RoboDK station: kr30 cnc 072119 yaaaasss.rdk

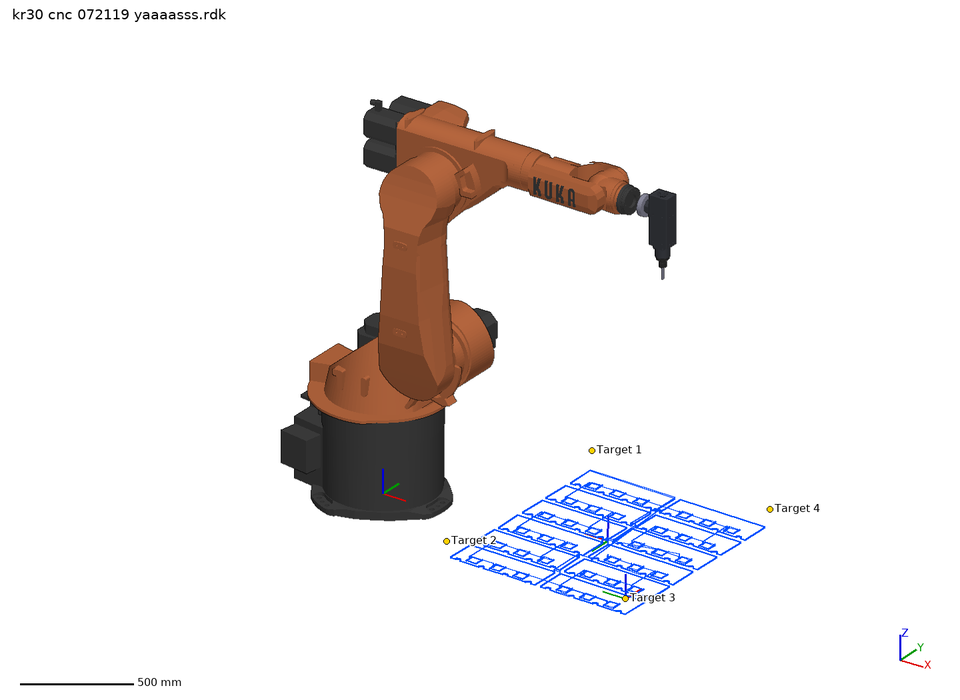
[picture v0: the station drawn from its stored meshes, robots at their saved joint values, targets as dots, program paths as lines]
Station kr30 cnc 072119 yaaaasss. Poses are relative to the parent item; angles as X-Y-Z fixed-axis rotations.
  - frame GIGASHEEN Base at (0, 0, 0) mm
    - robot GIGASHEEN (model KUKA KR 30 HA): 6 axes, payload 30 kg, reach 2033 mm, repeatability 0.05 mm, weight 665 kg
        modified DH rows (alpha deg, a mm, theta deg, d mm): 0, 0, 0, 815; -90, 350, 0, 0; 0, 850, -90, 0; -90, 145, 0, 820; 90, 0, 0, 0; -90, 0, 180, 170
        joint limits [-185, -135, -120, -350, -119, -350] to [185, 35, 158, 350, 119, 350]; home [0, -90, 90, 0, 0, 0]; saved at [0, -90, 90, 0, 0, 0]
      - tool 1/2" End Mill TCP, TCP at (337.71, -2.2, 160.57) mm, rotated rx 0 ry 90 rz 0 deg, size 415.8 x 102 x 153.6 mm
    - target Target 1 (joint target) at (982.46, 202.21, 406.25) mm, rotated rx -179.95 ry 0.15 rz -89.48 deg; joints [7.49, -59.642, 144.935, 97.969, -90.801, -4.608] of GIGASHEEN
    - target Target 2 (joint target) at (986.83, -921.64, 412.07) mm, rotated rx -179.94 ry 0.15 rz -89.48 deg; joints [51.766, -38.608, 94.384, 136.851, -116.554, -22.567] of GIGASHEEN
    - target Target 3 (joint target) at (1949.02, -919.97, 396.91) mm, rotated rx -179.94 ry 0.14 rz 179.61 deg; joints [29.5, -22.76, 62.288, 41.088, -47.759, -30.404] of GIGASHEEN
    - target Target 4 (joint target) at (1949.02, 190.94, 391.63) mm, rotated rx -179.94 ry 0.14 rz 179.61 deg; joints [-6.898, -35.989, 90.741, -8.88, -55.221, 5.167] of GIGASHEEN
  - machining project Machining Settings: C:/Users/liqui/OneDrive/Desktop/first half pipe jig.apt | rotZ(0) | rotX(0)*rotY(0) | rotZ(0)
  - program Prog2 (4 instructions, listed below)
  - frame Table at (1949.02, -919.97, 396.91) mm, rotated rx 0.87 ry 0.27 rz 90 deg
    - frame Frame 4 at (550, 480, -75) mm, rotated rx 0 ry 0 rz 90 deg
  - program Machining (1954 instructions, listed below)
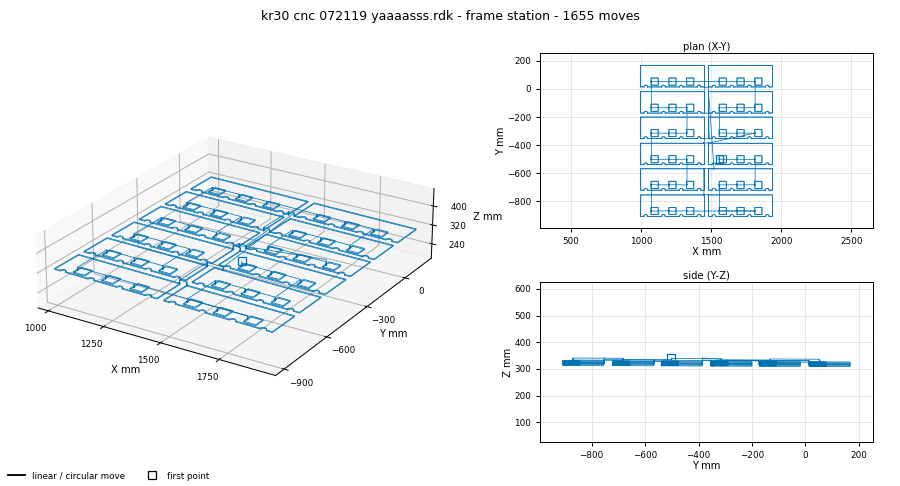
[picture p0: tool path of kr30 cnc 072119 yaaaasss.rdk in frame station, 1655 of 1659 moves have a stored position in this frame; points joined in program order, loops and branches not executed]

--- program Prog2 (robot GIGASHEEN) ---
  MoveJ (plywood back right safe) [its target is no longer in the station]
  MoveL (plywood back left safe) [its target is no longer in the station]
  MoveL (plywood front left safe) [its target is no longer in the station]
  MoveL (plywood front right safe) [its target is no longer in the station]

--- program Machining (robot GIGASHEEN) ---
  Smooth(1)
  Set Ref.: Frame 4
  Set Tool: 1/2" End Mill TCP
  Show 1/2" End Mill TCP
  Print: /'1001'
  Print: /''
  Print: /'2D Contour2'
  Set speed (1000.0 mm/s)
  MoveJ 1 to (-92.16, 131.48, 15) mm, rotated rx 180 ry 0 rz 0 deg; joints [21.959, -45.515, 117.936, 23.028, -72.87, -6.513]
  MoveL 2 to (-92.16, 131.48, 15) mm, rotated rx 180 ry 0 rz 0 deg; joints [21.959, -45.515, 117.936, 23.028, -72.87, -6.513]
  MoveL 3 to (-92.16, 131.48, 15) mm, rotated rx 180 ry 0 rz 0 deg; joints [21.959, -45.515, 117.936, 23.028, -72.87, -6.513]
  Set speed (1000.0 mm/s)
  MoveL 4 to (-92.16, 131.49, 6) mm, rotated rx -180 ry 0 rz 0 deg; joints [21.962, -44.952, 117.841, 22.976, -73.301, -6.323]
  Set speed (25.4 mm/s)
  MoveL 5 to (-92.16, 131.49, -3.54) mm, rotated rx -180 ry 0 rz 0 deg; joints [21.967, -44.354, 117.733, 22.924, -73.753, -6.125]
  MoveC 6 to (-91.98, 131.49, -3.99) mm, rotated rx -180 ry 0 rz 0 deg; joints [21.97, -44.331, 117.743, 22.924, -73.782, -6.113] to (-91.53, 131.48, -4.17) mm, rotated rx 180 ry 0 rz 0 deg; joints [21.977, -44.333, 117.775, 22.928, -73.811, -6.103]
  Set speed (50.8 mm/s)
  MoveL 7 to (-90.89, 131.48, -4.18) mm, rotated rx 180 ry 0 rz 0 deg; joints [21.987, -44.352, 117.824, 22.935, -73.84, -6.093]
  MoveC 8 to (-90.44, 131.3, -4.18) mm, rotated rx -180 ry 0 rz 0 deg; joints [21.987, -44.368, 117.865, 22.932, -73.863, -6.083] to (-90.26, 130.85, -4.18) mm, rotated rx -180 ry 0 rz 0 deg; joints [21.972, -44.379, 117.893, 22.915, -73.877, -6.072]
  MoveL 9 to (-90.26, 105.45, -4.17) mm, rotated rx -180 ry 0 rz 0 deg; joints [20.95, -44.663, 118.664, 21.805, -74.218, -5.605]
  MoveL 10 to (-141.06, 105.45, -4.17) mm, rotated rx -180 ry 0 rz 0 deg; joints [20.189, -43.084, 114.66, 21.285, -71.881, -6.316]
  MoveL 11 to (-141.06, 156.25, -4.17) mm, rotated rx -180 ry 0 rz 0 deg; joints [22.16, -42.482, 113.093, 23.47, -71.231, -7.326]
  MoveL 12 to (-90.26, 156.25, -4.17) mm, rotated rx 180 ry 0 rz 0 deg; joints [22.98, -44.078, 117.084, 24.017, -73.527, -6.56]
  MoveL 13 to (-90.26, 130.85, -4.18) mm, rotated rx -180 ry 0 rz 0 deg; joints [21.972, -44.379, 117.893, 22.915, -73.877, -6.072]
  MoveC 14 to (-90.44, 130.4, -4.17) mm, rotated rx -180 ry 0 rz 0 deg; joints [21.951, -44.379, 117.893, 22.893, -73.875, -6.066] to (-90.89, 130.21, -4.18) mm, rotated rx 180 ry 0 rz 0 deg; joints [21.937, -44.367, 117.864, 22.88, -73.857, -6.069]
  MoveL 15 to (-91.53, 130.21, -4.18) mm, rotated rx 180 ry 0 rz 0 deg; joints [21.926, -44.348, 117.815, 22.873, -73.829, -6.079]
  MoveC 16 to (-91.98, 130.21, -3.99) mm, rotated rx 180 ry 0 rz 0 deg; joints [21.919, -44.346, 117.782, 22.869, -73.8, -6.089] to (-92.16, 130.21, -3.54) mm, rotated rx -180 ry 0 rz 0 deg; joints [21.916, -44.368, 117.773, 22.869, -73.77, -6.101]
  Set speed (1000.0 mm/s)
  MoveL 17 to (-92.16, 130.21, 5) mm, rotated rx -180 ry 0 rz 0 deg; joints [21.912, -44.904, 117.87, 22.915, -73.365, -6.278]
  MoveL 18 to (-92.16, 131.48, 5) mm, rotated rx -180 ry 0 rz 0 deg; joints [21.963, -44.89, 117.83, 22.971, -73.348, -6.302]
  Set speed (25.4 mm/s)
  MoveL 19 to (-92.16, 131.49, 1.83) mm, rotated rx -180 ry 0 rz 0 deg; joints [21.964, -44.691, 117.795, 22.953, -73.499, -6.236]
  MoveL 20 to (-92.16, 131.49, -7.71) mm, rotated rx 180 ry 0 rz 0 deg; joints [21.968, -44.091, 117.684, 22.902, -73.949, -6.039]
  MoveC 21 to (-91.98, 131.48, -8.16) mm, rotated rx 180 ry 0 rz 0 deg; joints [21.972, -44.069, 117.693, 22.902, -73.979, -6.027] to (-91.53, 131.48, -8.35) mm, rotated rx 180 ry 0 rz 0 deg; joints [21.979, -44.07, 117.725, 22.906, -74.008, -6.017]
  Set speed (50.8 mm/s)
  MoveL 22 to (-90.89, 131.48, -8.35) mm, rotated rx 180 ry 0 rz 0 deg; joints [21.989, -44.089, 117.774, 22.913, -74.037, -6.007]
  MoveC 23 to (-90.44, 131.3, -8.35) mm, rotated rx 180 ry 0 rz 0 deg; joints [21.989, -44.105, 117.815, 22.91, -74.059, -5.997] to (-90.26, 130.85, -8.35) mm, rotated rx -180 ry 0 rz 0 deg; joints [21.974, -44.116, 117.843, 22.893, -74.074, -5.986]
  MoveL 24 to (-90.26, 105.45, -8.35) mm, rotated rx -180 ry 0 rz 0 deg; joints [20.951, -44.398, 118.614, 21.784, -74.418, -5.522]
  MoveL 25 to (-141.06, 105.45, -8.35) mm, rotated rx 180 ry 0 rz 0 deg; joints [20.191, -42.829, 114.611, 21.263, -72.072, -6.238]
  MoveL 26 to (-141.06, 156.25, -8.35) mm, rotated rx 180 ry 0 rz 0 deg; joints [22.162, -42.232, 113.044, 23.445, -71.416, -7.242]
  MoveL 27 to (-90.26, 156.25, -8.35) mm, rotated rx 180 ry 0 rz 0 deg; joints [22.982, -43.817, 117.034, 23.994, -73.72, -6.471]
  MoveL 28 to (-90.26, 130.85, -8.35) mm, rotated rx -180 ry 0 rz 0 deg; joints [21.974, -44.116, 117.843, 22.893, -74.074, -5.986]
  MoveC 29 to (-90.44, 130.4, -8.35) mm, rotated rx 180 ry 0 rz 0 deg; joints [21.953, -44.115, 117.843, 22.871, -74.072, -5.981] to (-90.89, 130.21, -8.35) mm, rotated rx 180 ry 0 rz 0 deg; joints [21.938, -44.104, 117.814, 22.858, -74.054, -5.984]
  MoveL 30 to (-91.53, 130.21, -8.35) mm, rotated rx 180 ry 0 rz 0 deg; joints [21.928, -44.085, 117.765, 22.851, -74.025, -5.993]
  MoveC 31 to (-91.98, 130.21, -8.16) mm, rotated rx -180 ry 0 rz 0 deg; joints [21.921, -44.083, 117.732, 22.847, -73.996, -6.004] to (-92.16, 130.22, -7.72) mm, rotated rx -180 ry 0 rz 0 deg; joints [21.918, -44.106, 117.723, 22.847, -73.966, -6.015]
  Set speed (1000.0 mm/s)
  MoveL 32 to (-92.16, 130.21, 6) mm, rotated rx -180 ry 0 rz 0 deg; joints [21.912, -44.967, 117.881, 22.921, -73.318, -6.299]
  MoveL 33 to (-219.16, 131.48, 6) mm, rotated rx 180 ry 0 rz 0 deg; joints [20.086, -40.721, 107.569, 21.82, -67.469, -8.132]
  Set speed (25.4 mm/s)
  MoveL 34 to (-219.16, 131.48, -3.54) mm, rotated rx -180 ry 0 rz 0 deg; joints [20.089, -40.181, 107.465, 21.757, -67.874, -7.958]
  MoveC 35 to (-218.98, 131.48, -3.99) mm, rotated rx 180 ry 0 rz 0 deg; joints [20.092, -40.162, 107.476, 21.756, -67.902, -7.948] to (-218.53, 131.49, -4.17) mm, rotated rx -180 ry 0 rz 0 deg; joints [20.098, -40.168, 107.512, 21.758, -67.931, -7.938]
  Set speed (50.8 mm/s)
  MoveL 36 to (-217.89, 131.48, -4.17) mm, rotated rx 180 ry 0 rz 0 deg; joints [20.107, -40.19, 107.565, 21.762, -67.962, -7.929]
  MoveC 37 to (-217.44, 131.3, -4.18) mm, rotated rx 180 ry 0 rz 0 deg; joints [20.106, -40.208, 107.609, 21.758, -67.985, -7.918] to (-217.26, 130.85, -4.18) mm, rotated rx -180 ry 0 rz 0 deg; joints [20.092, -40.22, 107.638, 21.74, -67.999, -7.906]
  MoveL 38 to (-217.26, 105.45, -4.18) mm, rotated rx 180 ry 0 rz 0 deg; joints [19.142, -40.524, 108.399, 20.66, -68.295, -7.365]
  MoveL 39 to (-268.06, 105.45, -4.18) mm, rotated rx 180 ry 0 rz 0 deg; joints [18.501, -38.685, 104.03, 20.345, -65.836, -8.068]
  MoveL 40 to (-268.06, 156.25, -4.18) mm, rotated rx -180 ry 0 rz 0 deg; joints [20.336, -38.042, 102.464, 22.49, -65.261, -9.235]
  MoveL 41 to (-217.26, 156.25, -4.17) mm, rotated rx -180 ry 0 rz 0 deg; joints [21.03, -39.899, 106.838, 22.816, -67.694, -8.465]
  MoveL 42 to (-217.26, 130.85, -4.18) mm, rotated rx -180 ry 0 rz 0 deg; joints [20.092, -40.22, 107.638, 21.74, -67.999, -7.906]
  MoveC 43 to (-217.44, 130.4, -4.18) mm, rotated rx -180 ry 0 rz 0 deg; joints [20.073, -40.219, 107.636, 21.719, -67.996, -7.899] to (-217.89, 130.21, -4.17) mm, rotated rx 180 ry 0 rz 0 deg; joints [20.06, -40.206, 107.604, 21.708, -67.977, -7.901]
  MoveL 44 to (-218.53, 130.21, -4.17) mm, rotated rx 180 ry 0 rz 0 deg; joints [20.051, -40.183, 107.551, 21.704, -67.946, -7.91]
  MoveC 45 to (-218.98, 130.21, -3.99) mm, rotated rx -180 ry 0 rz 0 deg; joints [20.045, -40.178, 107.515, 21.702, -67.917, -7.92] to (-219.16, 130.21, -3.54) mm, rotated rx 180 ry 0 rz 0 deg; joints [20.042, -40.197, 107.504, 21.703, -67.889, -7.931]
  Set speed (1000.0 mm/s)
  MoveL 46 to (-219.16, 130.21, 5) mm, rotated rx -180 ry 0 rz 0 deg; joints [20.039, -40.68, 107.597, 21.759, -67.527, -8.086]
  MoveL 47 to (-219.16, 131.48, 5) mm, rotated rx 180 ry 0 rz 0 deg; joints [20.086, -40.665, 107.558, 21.813, -67.512, -8.113]
  Set speed (25.4 mm/s)
  MoveL 48 to (-219.16, 131.48, 1.82) mm, rotated rx 180 ry 0 rz 0 deg; joints [20.087, -40.485, 107.524, 21.792, -67.647, -8.056]
  MoveL 49 to (-219.16, 131.48, -7.72) mm, rotated rx -180 ry 0 rz 0 deg; joints [20.091, -39.944, 107.417, 21.731, -68.05, -7.883]
  MoveC 50 to (-218.98, 131.48, -8.16) mm, rotated rx -180 ry 0 rz 0 deg; joints [20.094, -39.925, 107.428, 21.729, -68.078, -7.873] to (-218.53, 131.49, -8.35) mm, rotated rx -180 ry 0 rz 0 deg; joints [20.1, -39.931, 107.464, 21.731, -68.107, -7.863]
  Set speed (50.8 mm/s)
  MoveL 51 to (-217.89, 131.48, -8.35) mm, rotated rx -180 ry 0 rz 0 deg; joints [20.108, -39.953, 107.517, 21.736, -68.138, -7.854]
  MoveC 52 to (-217.44, 131.3, -8.35) mm, rotated rx 180 ry 0 rz 0 deg; joints [20.108, -39.971, 107.561, 21.731, -68.161, -7.843] to (-217.26, 130.85, -8.35) mm, rotated rx -180 ry 0 rz 0 deg; joints [20.094, -39.983, 107.59, 21.713, -68.176, -7.831]
  MoveL 53 to (-217.26, 105.45, -8.35) mm, rotated rx -180 ry 0 rz 0 deg; joints [19.144, -40.285, 108.351, 20.635, -68.474, -7.293]
  MoveL 54 to (-268.06, 105.45, -8.35) mm, rotated rx 180 ry 0 rz 0 deg; joints [18.502, -38.455, 103.982, 20.319, -66.007, -7.999]
  MoveL 55 to (-268.06, 156.25, -8.35) mm, rotated rx -180 ry 0 rz 0 deg; joints [20.338, -37.815, 102.416, 22.46, -65.427, -9.16]
  MoveL 56 to (-217.26, 156.25, -8.35) mm, rotated rx 180 ry 0 rz 0 deg; joints [21.032, -39.663, 106.79, 22.788, -67.868, -8.387]
  MoveL 57 to (-217.26, 130.85, -8.35) mm, rotated rx -180 ry 0 rz 0 deg; joints [20.094, -39.983, 107.59, 21.713, -68.176, -7.831]
  MoveC 58 to (-217.44, 130.4, -8.35) mm, rotated rx -180 ry 0 rz 0 deg; joints [20.074, -39.982, 107.588, 21.693, -68.172, -7.824] to (-217.89, 130.22, -8.35) mm, rotated rx -180 ry 0 rz 0 deg; joints [20.061, -39.968, 107.556, 21.682, -68.153, -7.826]
  MoveL 59 to (-218.53, 130.21, -8.35) mm, rotated rx -180 ry 0 rz 0 deg; joints [20.053, -39.946, 107.503, 21.677, -68.123, -7.835]
  MoveC 60 to (-218.98, 130.22, -8.16) mm, rotated rx -180 ry 0 rz 0 deg; joints [20.047, -39.941, 107.467, 21.675, -68.093, -7.845] to (-219.16, 130.21, -7.72) mm, rotated rx -180 ry 0 rz 0 deg; joints [20.044, -39.96, 107.456, 21.677, -68.066, -7.856]
  Set speed (1000.0 mm/s)
  MoveL 61 to (-219.16, 130.21, 6) mm, rotated rx 180 ry 0 rz 0 deg; joints [20.039, -40.737, 107.608, 21.766, -67.484, -8.104]
  MoveL 62 to (-346.16, 131.48, 6) mm, rotated rx -180 ry 0 rz 0 deg; joints [18.494, -35.82, 96.268, 21.203, -61.256, -10.004]
  Set speed (25.4 mm/s)
  MoveL 63 to (-346.16, 131.48, -3.54) mm, rotated rx 180 ry 0 rz 0 deg; joints [18.497, -35.327, 96.164, 21.13, -61.62, -9.846]
  MoveC 64 to (-345.98, 131.48, -3.99) mm, rotated rx -180 ry 0 rz 0 deg; joints [18.5, -35.311, 96.177, 21.127, -61.646, -9.836] to (-345.53, 131.48, -4.17) mm, rotated rx -180 ry 0 rz 0 deg; joints [18.505, -35.32, 96.217, 21.127, -61.676, -9.825]
  Set speed (50.8 mm/s)
  MoveL 65 to (-344.89, 131.48, -4.17) mm, rotated rx -180 ry 0 rz 0 deg; joints [18.512, -35.346, 96.277, 21.129, -61.709, -9.816]
  MoveC 66 to (-344.44, 131.3, -4.18) mm, rotated rx 180 ry 0 rz 0 deg; joints [18.511, -35.367, 96.325, 21.122, -61.734, -9.804] to (-344.26, 130.85, -4.18) mm, rotated rx 180 ry 0 rz 0 deg; joints [18.498, -35.381, 96.356, 21.103, -61.748, -9.79]
  MoveL 67 to (-344.26, 105.45, -4.17) mm, rotated rx -180 ry 0 rz 0 deg; joints [17.613, -35.708, 97.129, 20.031, -62.016, -9.159]
  MoveL 68 to (-395.06, 105.45, -4.18) mm, rotated rx -180 ry 0 rz 0 deg; joints [17.065, -33.559, 92.253, 19.936, -59.36, -9.934]
  MoveL 69 to (-395.06, 156.25, -4.17) mm, rotated rx -180 ry 0 rz 0 deg; joints [18.779, -32.861, 90.636, 22.094, -58.825, -11.299]
  MoveL 70 to (-344.26, 156.25, -4.17) mm, rotated rx 180 ry 0 rz 0 deg; joints [19.373, -35.034, 95.54, 22.176, -61.47, -10.439]
  MoveL 71 to (-344.26, 130.85, -4.18) mm, rotated rx 180 ry 0 rz 0 deg; joints [18.498, -35.381, 96.356, 21.103, -61.748, -9.79]
  MoveC 72 to (-344.44, 130.4, -4.18) mm, rotated rx -180 ry 0 rz 0 deg; joints [18.48, -35.379, 96.353, 21.084, -61.743, -9.781] to (-344.89, 130.21, -4.17) mm, rotated rx 180 ry 0 rz 0 deg; joints [18.468, -35.363, 96.316, 21.075, -61.722, -9.784]
  MoveL 73 to (-345.53, 130.21, -4.18) mm, rotated rx 180 ry 0 rz 0 deg; joints [18.461, -35.337, 96.257, 21.073, -61.69, -9.793]
  MoveC 74 to (-345.98, 130.21, -3.99) mm, rotated rx 180 ry 0 rz 0 deg; joints [18.456, -35.328, 96.217, 21.073, -61.66, -9.803] to (-346.16, 130.21, -3.54) mm, rotated rx -180 ry 0 rz 0 deg; joints [18.453, -35.344, 96.204, 21.076, -61.633, -9.814]
  Set speed (1000.0 mm/s)
  MoveL 75 to (-346.16, 130.21, 5) mm, rotated rx -180 ry 0 rz 0 deg; joints [18.451, -35.785, 96.297, 21.141, -61.307, -9.955]
  MoveL 76 to (-346.16, 131.48, 5) mm, rotated rx 180 ry 0 rz 0 deg; joints [18.494, -35.768, 96.257, 21.195, -61.294, -9.988]
  Set speed (25.4 mm/s)
  MoveL 77 to (-346.16, 131.49, 1.83) mm, rotated rx -180 ry 0 rz 0 deg; joints [18.496, -35.604, 96.223, 21.171, -61.415, -9.935]
  MoveL 78 to (-346.16, 131.48, -7.71) mm, rotated rx -180 ry 0 rz 0 deg; joints [18.499, -35.11, 96.117, 21.099, -61.778, -9.777]
  MoveC 79 to (-345.98, 131.48, -8.16) mm, rotated rx -180 ry 0 rz 0 deg; joints [18.501, -35.095, 96.129, 21.096, -61.804, -9.767] to (-345.53, 131.48, -8.35) mm, rotated rx 180 ry 0 rz 0 deg; joints [18.506, -35.103, 96.169, 21.096, -61.834, -9.757]
  Set speed (50.8 mm/s)
  MoveL 80 to (-344.89, 131.48, -8.35) mm, rotated rx -180 ry 0 rz 0 deg; joints [18.514, -35.129, 96.229, 21.097, -61.867, -9.747]
  MoveC 81 to (-344.44, 131.3, -8.35) mm, rotated rx -180 ry 0 rz 0 deg; joints [18.513, -35.15, 96.277, 21.091, -61.892, -9.735] to (-344.26, 130.85, -8.35) mm, rotated rx 180 ry 0 rz 0 deg; joints [18.499, -35.164, 96.308, 21.072, -61.906, -9.721]
  MoveL 82 to (-344.26, 105.45, -8.35) mm, rotated rx -180 ry 0 rz 0 deg; joints [17.614, -35.49, 97.082, 20.002, -62.177, -9.094]
  MoveL 83 to (-395.06, 105.45, -8.35) mm, rotated rx -180 ry 0 rz 0 deg; joints [17.067, -33.348, 92.205, 19.904, -59.513, -9.87]
  MoveL 84 to (-395.06, 156.25, -8.35) mm, rotated rx 180 ry 0 rz 0 deg; joints [18.78, -32.652, 90.588, 22.059, -58.974, -11.23]
  MoveL 85 to (-344.26, 156.25, -8.35) mm, rotated rx 180 ry 0 rz 0 deg; joints [19.375, -34.819, 95.493, 22.143, -61.625, -10.367]
  MoveL 86 to (-344.26, 130.85, -8.35) mm, rotated rx 180 ry 0 rz 0 deg; joints [18.499, -35.164, 96.308, 21.072, -61.906, -9.721]
  MoveC 87 to (-344.44, 130.4, -8.35) mm, rotated rx -180 ry 0 rz 0 deg; joints [18.481, -35.162, 96.305, 21.053, -61.902, -9.713] to (-344.89, 130.21, -8.35) mm, rotated rx -180 ry 0 rz 0 deg; joints [18.47, -35.146, 96.269, 21.044, -61.88, -9.715]
  MoveL 88 to (-345.53, 130.22, -8.35) mm, rotated rx -180 ry 0 rz 0 deg; joints [18.462, -35.12, 96.209, 21.042, -61.848, -9.725]
  MoveC 89 to (-345.98, 130.22, -8.16) mm, rotated rx -180 ry 0 rz 0 deg; joints [18.457, -35.111, 96.169, 21.042, -61.818, -9.735] to (-346.16, 130.21, -7.72) mm, rotated rx 180 ry 0 rz 0 deg; joints [18.455, -35.127, 96.157, 21.045, -61.791, -9.745]
  Set speed (1000.0 mm/s)
  MoveL 90 to (-346.16, 130.21, 6) mm, rotated rx -180 ry 0 rz 0 deg; joints [18.45, -35.837, 96.307, 21.149, -61.269, -9.972]
  MoveL 91 to (-346.16, 313.35, 6) mm, rotated rx -180 ry 0 rz 0 deg; joints [24.544, -32.855, 89.443, 28.944, -59.101, -15.185]
  Set speed (25.4 mm/s)
  MoveL 92 to (-346.16, 313.36, -3.54) mm, rotated rx -180 ry 0 rz 0 deg; joints [24.547, -32.384, 89.339, 28.843, -59.423, -14.981]
  MoveC 93 to (-345.98, 313.35, -3.99) mm, rotated rx 180 ry 0 rz 0 deg; joints [24.55, -32.37, 89.352, 28.838, -59.447, -14.968] to (-345.53, 313.35, -4.17) mm, rotated rx 180 ry 0 rz 0 deg; joints [24.557, -32.38, 89.393, 28.837, -59.476, -14.954]
  Set speed (50.8 mm/s)
  MoveL 94 to (-344.89, 313.35, -4.18) mm, rotated rx -180 ry 0 rz 0 deg; joints [24.566, -32.408, 89.454, 28.838, -59.508, -14.94]
  MoveC 95 to (-344.44, 313.17, -4.17) mm, rotated rx -180 ry 0 rz 0 deg; joints [24.566, -32.431, 89.506, 28.83, -59.533, -14.924] to (-344.26, 312.72, -4.18) mm, rotated rx -180 ry 0 rz 0 deg; joints [24.555, -32.447, 89.543, 28.811, -59.549, -14.906]
  MoveL 96 to (-344.26, 287.32, -4.18) mm, rotated rx -180 ry 0 rz 0 deg; joints [23.74, -32.923, 90.634, 27.729, -59.883, -14.121]
  MoveL 97 to (-395.06, 287.32, -4.17) mm, rotated rx -180 ry 0 rz 0 deg; joints [23.039, -30.666, 85.619, 27.719, -57.26, -15.221]
  MoveL 98 to (-395.06, 338.12, -4.17) mm, rotated rx -180 ry 0 rz 0 deg; joints [24.622, -29.649, 83.326, 29.933, -56.588, -16.922]
  MoveL 99 to (-344.26, 338.12, -4.17) mm, rotated rx -180 ry 0 rz 0 deg; joints [25.359, -31.949, 88.405, 29.898, -59.207, -15.718]
  MoveL 100 to (-344.26, 312.72, -4.18) mm, rotated rx -180 ry 0 rz 0 deg; joints [24.555, -32.447, 89.543, 28.811, -59.549, -14.906]
  MoveC 101 to (-344.44, 312.27, -4.17) mm, rotated rx -180 ry 0 rz 0 deg; joints [24.538, -32.448, 89.545, 28.792, -59.545, -14.896] to (-344.89, 312.08, -4.17) mm, rotated rx 180 ry 0 rz 0 deg; joints [24.525, -32.432, 89.51, 28.783, -59.525, -14.9]
  MoveL 102 to (-345.53, 312.08, -4.18) mm, rotated rx 180 ry 0 rz 0 deg; joints [24.516, -32.405, 89.449, 28.783, -59.493, -14.914]
  MoveC 103 to (-345.98, 312.08, -3.99) mm, rotated rx -180 ry 0 rz 0 deg; joints [24.51, -32.394, 89.408, 28.784, -59.464, -14.928] to (-346.16, 312.08, -3.54) mm, rotated rx 180 ry 0 rz 0 deg; joints [24.507, -32.409, 89.395, 28.789, -59.44, -14.941]
  Set speed (1000.0 mm/s)
  MoveL 104 to (-346.16, 312.09, 5) mm, rotated rx -180 ry 0 rz 0 deg; joints [24.503, -32.831, 89.489, 28.879, -59.151, -15.123]
  MoveL 105 to (-346.16, 313.35, 5) mm, rotated rx -180 ry 0 rz 0 deg; joints [24.544, -32.806, 89.433, 28.933, -59.135, -15.164]
  Set speed (25.4 mm/s)
  MoveL 106 to (-346.16, 313.36, 1.82) mm, rotated rx -180 ry 0 rz 0 deg; joints [24.545, -32.65, 89.399, 28.899, -59.242, -15.095]
  MoveL 107 to (-346.16, 313.35, -7.71) mm, rotated rx -180 ry 0 rz 0 deg; joints [24.549, -32.177, 89.291, 28.799, -59.563, -14.893]
  MoveC 108 to (-345.98, 313.36, -8.16) mm, rotated rx -180 ry 0 rz 0 deg; joints [24.552, -32.163, 89.303, 28.795, -59.587, -14.879] to (-345.53, 313.35, -8.35) mm, rotated rx 180 ry 0 rz 0 deg; joints [24.558, -32.173, 89.345, 28.794, -59.616, -14.866]
  Set speed (50.8 mm/s)
  MoveL 109 to (-344.89, 313.35, -8.35) mm, rotated rx -180 ry 0 rz 0 deg; joints [24.567, -32.2, 89.406, 28.794, -59.648, -14.852]
  MoveC 110 to (-344.44, 313.17, -8.35) mm, rotated rx 180 ry 0 rz 0 deg; joints [24.568, -32.223, 89.457, 28.787, -59.673, -14.836] to (-344.26, 312.72, -8.35) mm, rotated rx -180 ry 0 rz 0 deg; joints [24.556, -32.24, 89.495, 28.768, -59.689, -14.818]
  MoveL 111 to (-344.26, 287.32, -8.35) mm, rotated rx -180 ry 0 rz 0 deg; joints [23.741, -32.714, 90.586, 27.687, -60.025, -14.035]
  MoveL 112 to (-395.06, 287.32, -8.35) mm, rotated rx -180 ry 0 rz 0 deg; joints [23.04, -30.463, 85.57, 27.675, -57.397, -15.137]
  MoveL 113 to (-395.06, 338.12, -8.35) mm, rotated rx 180 ry 0 rz 0 deg; joints [24.624, -29.449, 83.277, 29.886, -56.719, -16.832]
  MoveL 114 to (-344.26, 338.12, -8.35) mm, rotated rx -180 ry 0 rz 0 deg; joints [25.361, -31.743, 88.356, 29.853, -59.344, -15.627]
  MoveL 115 to (-344.26, 312.72, -8.35) mm, rotated rx -180 ry 0 rz 0 deg; joints [24.556, -32.24, 89.495, 28.768, -59.689, -14.818]
  MoveC 116 to (-344.44, 312.27, -8.35) mm, rotated rx 180 ry 0 rz 0 deg; joints [24.539, -32.24, 89.497, 28.749, -59.685, -14.808] to (-344.89, 312.09, -8.35) mm, rotated rx -180 ry 0 rz 0 deg; joints [24.527, -32.225, 89.462, 28.74, -59.665, -14.812]
  MoveL 117 to (-345.53, 312.08, -8.35) mm, rotated rx 180 ry 0 rz 0 deg; joints [24.518, -32.197, 89.4, 28.739, -59.633, -14.826]
  MoveC 118 to (-345.98, 312.08, -8.16) mm, rotated rx -180 ry 0 rz 0 deg; joints [24.511, -32.187, 89.359, 28.741, -59.604, -14.84] to (-346.16, 312.08, -7.72) mm, rotated rx -180 ry 0 rz 0 deg; joints [24.508, -32.201, 89.347, 28.745, -59.58, -14.853]
  Set speed (1000.0 mm/s)
  MoveL 119 to (-346.16, 312.09, 6) mm, rotated rx -180 ry 0 rz 0 deg; joints [24.503, -32.88, 89.499, 28.89, -59.118, -15.145]
  MoveL 120 to (-219.16, 313.36, 6) mm, rotated rx 180 ry 0 rz 0 deg; joints [26.529, -37.966, 100.93, 29.478, -65.154, -12.654]
  Set speed (25.4 mm/s)
  MoveL 121 to (-219.16, 313.35, -3.54) mm, rotated rx -180 ry 0 rz 0 deg; joints [26.533, -37.456, 100.827, 29.39, -65.51, -12.436]
  MoveC 122 to (-218.98, 313.35, -3.99) mm, rotated rx -180 ry 0 rz 0 deg; joints [26.537, -37.439, 100.838, 29.387, -65.535, -12.422] to (-218.53, 313.35, -4.17) mm, rotated rx -180 ry 0 rz 0 deg; joints [26.544, -37.445, 100.874, 29.389, -65.563, -12.409]
  Set speed (50.8 mm/s)
  MoveL 123 to (-217.89, 313.36, -4.18) mm, rotated rx -180 ry 0 rz 0 deg; joints [26.555, -37.468, 100.928, 29.394, -65.592, -12.397]
  MoveC 124 to (-217.44, 313.17, -4.18) mm, rotated rx -180 ry 0 rz 0 deg; joints [26.556, -37.488, 100.974, 29.389, -65.615, -12.384] to (-217.26, 312.72, -4.18) mm, rotated rx -180 ry 0 rz 0 deg; joints [26.544, -37.503, 101.009, 29.372, -65.63, -12.368]
  MoveL 125 to (-217.26, 287.32, -4.17) mm, rotated rx -180 ry 0 rz 0 deg; joints [25.681, -37.942, 102.061, 28.315, -65.983, -11.678]
  MoveL 126 to (-268.06, 287.32, -4.18) mm, rotated rx -180 ry 0 rz 0 deg; joints [24.87, -36.03, 97.657, 27.993, -63.611, -12.617]
  MoveL 127 to (-268.06, 338.12, -4.18) mm, rotated rx -180 ry 0 rz 0 deg; joints [26.545, -35.106, 95.487, 30.12, -62.917, -14.089]
  MoveL 128 to (-217.26, 338.12, -4.18) mm, rotated rx 180 ry 0 rz 0 deg; joints [27.394, -37.044, 99.914, 30.427, -65.27, -13.082]
  MoveL 129 to (-217.26, 312.72, -4.18) mm, rotated rx -180 ry 0 rz 0 deg; joints [26.544, -37.503, 101.009, 29.372, -65.63, -12.368]
  MoveC 130 to (-217.44, 312.27, -4.17) mm, rotated rx -180 ry 0 rz 0 deg; joints [26.526, -37.504, 101.012, 29.352, -65.627, -12.359] to (-217.89, 312.08, -4.18) mm, rotated rx 180 ry 0 rz 0 deg; joints [26.512, -37.491, 100.982, 29.341, -65.61, -12.362]
  MoveL 131 to (-218.53, 312.08, -4.18) mm, rotated rx -180 ry 0 rz 0 deg; joints [26.501, -37.468, 100.928, 29.336, -65.58, -12.374]
  MoveC 132 to (-218.98, 312.08, -3.99) mm, rotated rx 180 ry 0 rz 0 deg; joints [26.494, -37.461, 100.892, 29.335, -65.553, -12.387] to (-219.16, 312.08, -3.54) mm, rotated rx -180 ry 0 rz 0 deg; joints [26.49, -37.478, 100.881, 29.337, -65.528, -12.401]
  Set speed (1000.0 mm/s)
  MoveL 133 to (-219.16, 312.08, 5) mm, rotated rx -180 ry 0 rz 0 deg; joints [26.487, -37.935, 100.973, 29.415, -65.209, -12.596]
  MoveL 134 to (-219.16, 313.35, 5) mm, rotated rx -180 ry 0 rz 0 deg; joints [26.53, -37.913, 100.919, 29.468, -65.192, -12.631]
  Set speed (25.4 mm/s)
  MoveL 135 to (-219.16, 313.35, 1.82) mm, rotated rx -180 ry 0 rz 0 deg; joints [26.531, -37.743, 100.886, 29.439, -65.31, -12.558]
  MoveL 136 to (-219.16, 313.36, -7.71) mm, rotated rx -180 ry 0 rz 0 deg; joints [26.535, -37.232, 100.78, 29.353, -65.665, -12.341]
  MoveC 137 to (-218.98, 313.35, -8.16) mm, rotated rx -180 ry 0 rz 0 deg; joints [26.538, -37.214, 100.791, 29.35, -65.69, -12.328] to (-218.53, 313.35, -8.35) mm, rotated rx -180 ry 0 rz 0 deg; joints [26.546, -37.221, 100.827, 29.352, -65.717, -12.315]
  Set speed (50.8 mm/s)
  MoveL 138 to (-217.89, 313.35, -8.35) mm, rotated rx 180 ry 0 rz 0 deg; joints [26.557, -37.244, 100.881, 29.356, -65.746, -12.303]
  MoveC 139 to (-217.44, 313.17, -8.35) mm, rotated rx -180 ry 0 rz 0 deg; joints [26.558, -37.264, 100.927, 29.352, -65.769, -12.289] to (-217.26, 312.72, -8.35) mm, rotated rx -180 ry 0 rz 0 deg; joints [26.546, -37.278, 100.961, 29.334, -65.784, -12.273]
  MoveL 140 to (-217.26, 287.32, -8.35) mm, rotated rx -180 ry 0 rz 0 deg; joints [25.683, -37.715, 102.014, 28.279, -66.141, -11.586]
  MoveL 141 to (-268.06, 287.32, -8.35) mm, rotated rx -180 ry 0 rz 0 deg; joints [24.872, -35.811, 97.609, 27.955, -63.763, -12.528]
  MoveL 142 to (-268.06, 338.12, -8.35) mm, rotated rx 180 ry 0 rz 0 deg; joints [26.547, -34.89, 95.44, 30.079, -63.063, -13.995]
  MoveL 143 to (-217.26, 338.12, -8.35) mm, rotated rx 180 ry 0 rz 0 deg; joints [27.396, -36.821, 99.867, 30.388, -65.421, -12.985]
  MoveL 144 to (-217.26, 312.72, -8.35) mm, rotated rx -180 ry 0 rz 0 deg; joints [26.546, -37.278, 100.961, 29.334, -65.784, -12.273]
  MoveC 145 to (-217.44, 312.27, -8.35) mm, rotated rx -180 ry 0 rz 0 deg; joints [26.528, -37.28, 100.964, 29.314, -65.782, -12.265] to (-217.89, 312.08, -8.35) mm, rotated rx -180 ry 0 rz 0 deg; joints [26.514, -37.266, 100.934, 29.303, -65.764, -12.268]
  MoveL 146 to (-218.53, 312.08, -8.35) mm, rotated rx -180 ry 0 rz 0 deg; joints [26.503, -37.243, 100.88, 29.299, -65.735, -12.28]
  MoveC 147 to (-218.98, 312.08, -8.16) mm, rotated rx -180 ry 0 rz 0 deg; joints [26.496, -37.237, 100.844, 29.297, -65.708, -12.293] to (-219.16, 312.08, -7.72) mm, rotated rx 180 ry 0 rz 0 deg; joints [26.492, -37.254, 100.834, 29.3, -65.683, -12.306]
  Set speed (1000.0 mm/s)
  MoveL 148 to (-219.16, 312.08, 6) mm, rotated rx 180 ry 0 rz 0 deg; joints [26.487, -37.989, 100.983, 29.425, -65.172, -12.619]
  MoveL 149 to (-92.16, 313.35, 6) mm, rotated rx -180 ry 0 rz 0 deg; joints [28.835, -42.353, 111.181, 30.723, -70.7, -10.362]
  Set speed (25.4 mm/s)
  MoveL 150 to (-92.16, 313.35, -3.54) mm, rotated rx 180 ry 0 rz 0 deg; joints [28.84, -41.795, 111.076, 30.647, -71.091, -10.118]
  MoveC 151 to (-91.98, 313.36, -3.99) mm, rotated rx -180 ry 0 rz 0 deg; joints [28.843, -41.774, 111.085, 30.646, -71.117, -10.104] to (-91.53, 313.36, -4.17) mm, rotated rx -180 ry 0 rz 0 deg; joints [28.852, -41.778, 111.118, 30.65, -71.144, -10.091]
  Set speed (50.8 mm/s)
  MoveL 152 to (-90.89, 313.35, -4.18) mm, rotated rx -180 ry 0 rz 0 deg; joints [28.865, -41.798, 111.166, 30.658, -71.17, -10.079]
  MoveC 153 to (-90.44, 313.17, -4.18) mm, rotated rx -180 ry 0 rz 0 deg; joints [28.867, -41.815, 111.209, 30.656, -71.192, -10.067] to (-90.26, 312.72, -4.18) mm, rotated rx 180 ry 0 rz 0 deg; joints [28.855, -41.828, 111.242, 30.64, -71.207, -10.052]
  MoveL 154 to (-90.26, 287.32, -4.17) mm, rotated rx -180 ry 0 rz 0 deg; joints [27.941, -42.241, 112.29, 29.583, -71.599, -9.426]
  MoveL 155 to (-141.06, 287.32, -4.18) mm, rotated rx 180 ry 0 rz 0 deg; joints [26.995, -40.599, 108.32, 28.998, -69.402, -10.319]
  MoveL 156 to (-141.06, 338.12, -4.18) mm, rotated rx -180 ry 0 rz 0 deg; joints [28.766, -39.735, 106.186, 31.103, -68.648, -11.639]
  MoveL 157 to (-90.26, 338.12, -4.17) mm, rotated rx 180 ry 0 rz 0 deg; joints [29.752, -41.397, 110.154, 31.69, -70.811, -10.701]
  MoveL 158 to (-90.26, 312.72, -4.18) mm, rotated rx 180 ry 0 rz 0 deg; joints [28.855, -41.828, 111.242, 30.64, -71.207, -10.052]
  MoveC 159 to (-90.44, 312.27, -4.17) mm, rotated rx -180 ry 0 rz 0 deg; joints [28.835, -41.83, 111.246, 30.619, -71.206, -10.044] to (-90.89, 312.08, -4.18) mm, rotated rx 180 ry 0 rz 0 deg; joints [28.82, -41.819, 111.22, 30.606, -71.19, -10.047]
  MoveL 160 to (-91.53, 312.08, -4.18) mm, rotated rx -180 ry 0 rz 0 deg; joints [28.807, -41.799, 111.171, 30.598, -71.163, -10.059]
  MoveC 161 to (-91.98, 312.08, -3.99) mm, rotated rx 180 ry 0 rz 0 deg; joints [28.798, -41.795, 111.139, 30.593, -71.137, -10.072] to (-92.16, 312.08, -3.54) mm, rotated rx -180 ry 0 rz 0 deg; joints [28.794, -41.816, 111.13, 30.595, -71.11, -10.086]
  Set speed (1000.0 mm/s)
  MoveL 162 to (-92.16, 312.08, 5) mm, rotated rx 180 ry 0 rz 0 deg; joints [28.79, -42.316, 111.224, 30.662, -70.76, -10.304]
  MoveL 163 to (-92.16, 313.35, 5) mm, rotated rx 180 ry 0 rz 0 deg; joints [28.836, -42.294, 111.17, 30.715, -70.741, -10.336]
  Set speed (25.4 mm/s)
  MoveL 164 to (-92.16, 313.36, 1.82) mm, rotated rx 180 ry 0 rz 0 deg; joints [28.837, -42.109, 111.136, 30.689, -70.871, -10.255]
  MoveL 165 to (-92.16, 313.35, -7.71) mm, rotated rx 180 ry 0 rz 0 deg; joints [28.842, -41.55, 111.028, 30.615, -71.261, -10.013]
  MoveC 166 to (-91.98, 313.35, -8.16) mm, rotated rx -180 ry 0 rz 0 deg; joints [28.845, -41.529, 111.037, 30.614, -71.287, -9.998] to (-91.53, 313.35, -8.35) mm, rotated rx -180 ry 0 rz 0 deg; joints [28.854, -41.532, 111.07, 30.618, -71.313, -9.985]
  Set speed (50.8 mm/s)
  MoveL 167 to (-90.89, 313.35, -8.35) mm, rotated rx -180 ry 0 rz 0 deg; joints [28.867, -41.552, 111.118, 30.626, -71.34, -9.974]
  MoveC 168 to (-90.44, 313.17, -8.35) mm, rotated rx -180 ry 0 rz 0 deg; joints [28.869, -41.569, 111.16, 30.624, -71.362, -9.961] to (-90.26, 312.72, -8.35) mm, rotated rx -180 ry 0 rz 0 deg; joints [28.857, -41.583, 111.194, 30.608, -71.377, -9.947]
  MoveL 169 to (-90.26, 287.32, -8.35) mm, rotated rx -180 ry 0 rz 0 deg; joints [27.943, -41.993, 112.242, 29.553, -71.773, -9.323]
  MoveL 170 to (-141.06, 287.32, -8.35) mm, rotated rx 180 ry 0 rz 0 deg; joints [26.996, -40.36, 108.273, 28.965, -69.569, -10.221]
  MoveL 171 to (-141.06, 338.12, -8.35) mm, rotated rx 180 ry 0 rz 0 deg; joints [28.768, -39.5, 106.139, 31.067, -68.808, -11.537]
  MoveL 172 to (-90.26, 338.12, -8.35) mm, rotated rx -180 ry 0 rz 0 deg; joints [29.754, -41.154, 110.106, 31.656, -70.977, -10.594]
  MoveL 173 to (-90.26, 312.72, -8.35) mm, rotated rx -180 ry 0 rz 0 deg; joints [28.857, -41.583, 111.194, 30.608, -71.377, -9.947]
  MoveC 174 to (-90.44, 312.27, -8.35) mm, rotated rx 180 ry 0 rz 0 deg; joints [28.837, -41.584, 111.198, 30.587, -71.376, -9.939] to (-90.89, 312.08, -8.35) mm, rotated rx 180 ry 0 rz 0 deg; joints [28.822, -41.573, 111.172, 30.574, -71.36, -9.942]
  MoveL 175 to (-91.53, 312.08, -8.35) mm, rotated rx 180 ry 0 rz 0 deg; joints [28.809, -41.553, 111.123, 30.566, -71.333, -9.954]
  MoveC 176 to (-91.98, 312.08, -8.16) mm, rotated rx 180 ry 0 rz 0 deg; joints [28.8, -41.55, 111.091, 30.561, -71.307, -9.966] to (-92.16, 312.08, -7.72) mm, rotated rx -180 ry 0 rz 0 deg; joints [28.796, -41.571, 111.082, 30.562, -71.28, -9.981]
  Set speed (1000.0 mm/s)
  MoveL 177 to (-92.16, 312.08, 6) mm, rotated rx 180 ry 0 rz 0 deg; joints [28.79, -42.374, 111.234, 30.67, -70.719, -10.33]
  MoveL 178 to (-92.16, 499.69, 6) mm, rotated rx -180 ry 0 rz 0 deg; joints [35.048, -38.673, 102.259, 38.322, -67.806, -15.742]
  Set speed (25.4 mm/s)
  MoveL 179 to (-92.16, 499.69, -3.54) mm, rotated rx 180 ry 0 rz 0 deg; joints [35.053, -38.157, 102.157, 38.224, -68.131, -15.468]
  MoveC 180 to (-91.98, 499.69, -3.99) mm, rotated rx -180 ry 0 rz 0 deg; joints [35.057, -38.139, 102.166, 38.221, -68.154, -15.451] to (-91.53, 499.69, -4.17) mm, rotated rx 180 ry 0 rz 0 deg; joints [35.067, -38.144, 102.199, 38.225, -68.178, -15.436]
  Set speed (50.8 mm/s)
  MoveL 181 to (-90.89, 499.69, -4.18) mm, rotated rx 180 ry 0 rz 0 deg; joints [35.081, -38.165, 102.247, 38.232, -68.204, -15.423]
  MoveC 182 to (-90.44, 499.51, -4.17) mm, rotated rx -180 ry 0 rz 0 deg; joints [35.085, -38.184, 102.292, 38.23, -68.225, -15.407] to (-90.26, 499.06, -4.17) mm, rotated rx 180 ry 0 rz 0 deg; joints [35.075, -38.201, 102.33, 38.214, -68.24, -15.389]
  MoveL 183 to (-90.26, 473.66, -4.17) mm, rotated rx -180 ry 0 rz 0 deg; joints [34.277, -38.76, 103.675, 37.196, -68.65, -14.581]
  MoveL 184 to (-141.06, 473.66, -4.17) mm, rotated rx -180 ry 0 rz 0 deg; joints [33.208, -37.034, 99.687, 36.642, -66.558, -15.642]
  MoveL 185 to (-141.06, 524.46, -4.18) mm, rotated rx -180 ry 0 rz 0 deg; joints [34.767, -35.864, 96.933, 38.702, -65.755, -17.336]
  MoveL 186 to (-90.26, 524.46, -4.17) mm, rotated rx -180 ry 0 rz 0 deg; joints [35.858, -37.619, 100.943, 39.229, -67.828, -16.224]
  MoveL 187 to (-90.26, 499.06, -4.17) mm, rotated rx 180 ry 0 rz 0 deg; joints [35.075, -38.201, 102.33, 38.214, -68.24, -15.389]
  MoveC 188 to (-90.44, 498.61, -4.17) mm, rotated rx -180 ry 0 rz 0 deg; joints [35.057, -38.204, 102.34, 38.194, -68.239, -15.378] to (-90.89, 498.42, -4.18) mm, rotated rx 180 ry 0 rz 0 deg; joints [35.041, -38.194, 102.316, 38.181, -68.224, -15.382]
  MoveL 189 to (-91.53, 498.42, -4.18) mm, rotated rx 180 ry 0 rz 0 deg; joints [35.027, -38.173, 102.267, 38.174, -68.199, -15.395]
  MoveC 190 to (-91.98, 498.42, -3.99) mm, rotated rx -180 ry 0 rz 0 deg; joints [35.018, -38.168, 102.234, 38.17, -68.174, -15.41] to (-92.16, 498.42, -3.54) mm, rotated rx 180 ry 0 rz 0 deg; joints [35.013, -38.186, 102.225, 38.173, -68.152, -15.426]
  Set speed (1000.0 mm/s)
  MoveL 191 to (-92.16, 498.42, 5) mm, rotated rx 180 ry 0 rz 0 deg; joints [35.009, -38.648, 102.317, 38.261, -67.86, -15.672]
  MoveL 192 to (-92.16, 499.69, 5) mm, rotated rx -180 ry 0 rz 0 deg; joints [35.049, -38.619, 102.249, 38.312, -67.84, -15.713]
  Set speed (25.4 mm/s)
  MoveL 193 to (-92.16, 499.69, 1.82) mm, rotated rx 180 ry 0 rz 0 deg; joints [35.05, -38.447, 102.215, 38.279, -67.948, -15.621]
  MoveL 194 to (-92.16, 499.69, -7.72) mm, rotated rx -180 ry 0 rz 0 deg; joints [35.055, -37.931, 102.11, 38.181, -68.273, -15.349]
  MoveC 195 to (-91.98, 499.69, -8.16) mm, rotated rx 180 ry 0 rz 0 deg; joints [35.059, -37.913, 102.119, 38.179, -68.295, -15.332] to (-91.53, 499.69, -8.35) mm, rotated rx -180 ry 0 rz 0 deg; joints [35.069, -37.918, 102.151, 38.182, -68.32, -15.317]
  Set speed (50.8 mm/s)
  MoveL 196 to (-90.89, 499.69, -8.35) mm, rotated rx -180 ry 0 rz 0 deg; joints [35.083, -37.939, 102.2, 38.19, -68.345, -15.304]
  MoveC 197 to (-90.44, 499.51, -8.35) mm, rotated rx -180 ry 0 rz 0 deg; joints [35.087, -37.958, 102.245, 38.188, -68.366, -15.289] to (-90.26, 499.06, -8.35) mm, rotated rx 180 ry 0 rz 0 deg; joints [35.077, -37.974, 102.283, 38.172, -68.381, -15.27]
  MoveL 198 to (-90.26, 473.66, -8.35) mm, rotated rx -180 ry 0 rz 0 deg; joints [34.279, -38.531, 103.627, 37.156, -68.796, -14.463]
  MoveL 199 to (-141.06, 473.66, -8.35) mm, rotated rx -180 ry 0 rz 0 deg; joints [33.21, -36.812, 99.639, 36.599, -66.699, -15.529]
  MoveL 200 to (-141.06, 524.46, -8.35) mm, rotated rx -180 ry 0 rz 0 deg; joints [34.769, -35.646, 96.886, 38.656, -65.889, -17.22]
  MoveL 201 to (-90.26, 524.46, -8.35) mm, rotated rx -180 ry 0 rz 0 deg; joints [35.86, -37.394, 100.896, 39.185, -67.966, -16.104]
  MoveL 202 to (-90.26, 499.06, -8.35) mm, rotated rx 180 ry 0 rz 0 deg; joints [35.077, -37.974, 102.283, 38.172, -68.381, -15.27]
  MoveC 203 to (-90.44, 498.61, -8.35) mm, rotated rx 180 ry 0 rz 0 deg; joints [35.059, -37.978, 102.293, 38.152, -68.381, -15.26] to (-90.89, 498.42, -8.35) mm, rotated rx 180 ry 0 rz 0 deg; joints [35.043, -37.967, 102.268, 38.139, -68.366, -15.263]
  MoveL 204 to (-91.53, 498.42, -8.35) mm, rotated rx -180 ry 0 rz 0 deg; joints [35.029, -37.946, 102.22, 38.132, -68.34, -15.276]
  MoveC 205 to (-91.98, 498.42, -8.16) mm, rotated rx -180 ry 0 rz 0 deg; joints [35.02, -37.941, 102.187, 38.128, -68.316, -15.291] to (-92.16, 498.42, -7.72) mm, rotated rx -180 ry 0 rz 0 deg; joints [35.015, -37.959, 102.178, 38.13, -68.293, -15.308]
  Set speed (1000.0 mm/s)
  MoveL 206 to (-92.16, 498.42, 6) mm, rotated rx -180 ry 0 rz 0 deg; joints [35.009, -38.702, 102.327, 38.271, -67.826, -15.701]
  MoveL 207 to (-219.16, 499.69, 6) mm, rotated rx 180 ry 0 rz 0 deg; joints [32.459, -34.052, 91.855, 37.24, -62.458, -18.541]
  Set speed (25.4 mm/s)
  MoveL 208 to (-219.16, 499.69, -3.54) mm, rotated rx 180 ry 0 rz 0 deg; joints [32.463, -33.574, 91.752, 37.127, -62.758, -18.288]
  MoveC 209 to (-218.98, 499.69, -3.99) mm, rotated rx -180 ry 0 rz 0 deg; joints [32.467, -33.559, 91.763, 37.122, -62.78, -18.271] to (-218.53, 499.69, -4.17) mm, rotated rx -180 ry 0 rz 0 deg; joints [32.475, -33.567, 91.8, 37.123, -62.806, -18.256]
  Set speed (50.8 mm/s)
  MoveL 210 to (-217.89, 499.69, -4.17) mm, rotated rx -180 ry 0 rz 0 deg; joints [32.487, -33.592, 91.856, 37.126, -62.834, -18.241]
  MoveC 211 to (-217.44, 499.51, -4.18) mm, rotated rx -180 ry 0 rz 0 deg; joints [32.49, -33.614, 91.905, 37.121, -62.857, -18.223] to (-217.26, 499.06, -4.17) mm, rotated rx -180 ry 0 rz 0 deg; joints [32.48, -33.632, 91.946, 37.103, -62.872, -18.203]
  MoveL 212 to (-217.26, 473.66, -4.18) mm, rotated rx -180 ry 0 rz 0 deg; joints [31.712, -34.232, 93.328, 36.047, -63.262, -17.321]
  MoveL 213 to (-268.06, 473.66, -4.17) mm, rotated rx -180 ry 0 rz 0 deg; joints [30.781, -32.203, 88.797, 35.823, -60.945, -18.528]
  MoveL 214 to (-268.06, 524.46, -4.17) mm, rotated rx 180 ry 0 rz 0 deg; joints [32.28, -30.934, 85.923, 37.987, -60.168, -20.409]
  MoveL 215 to (-217.26, 524.46, -4.17) mm, rotated rx -180 ry 0 rz 0 deg; joints [33.236, -33.008, 90.516, 38.162, -62.478, -19.115]
  MoveL 216 to (-217.26, 499.06, -4.18) mm, rotated rx -180 ry 0 rz 0 deg; joints [32.48, -33.632, 91.946, 37.103, -62.872, -18.203]
  MoveC 217 to (-217.44, 498.61, -4.18) mm, rotated rx -180 ry 0 rz 0 deg; joints [32.463, -33.636, 91.955, 37.083, -62.871, -18.192] to (-217.89, 498.42, -4.17) mm, rotated rx -180 ry 0 rz 0 deg; joints [32.449, -33.623, 91.926, 37.073, -62.854, -18.196]
  MoveL 218 to (-218.53, 498.42, -4.18) mm, rotated rx -180 ry 0 rz 0 deg; joints [32.437, -33.598, 91.871, 37.07, -62.825, -18.211]
  MoveC 219 to (-218.98, 498.42, -3.99) mm, rotated rx 180 ry 0 rz 0 deg; joints [32.428, -33.59, 91.834, 37.07, -62.799, -18.226] to (-219.16, 498.42, -3.54) mm, rotated rx -180 ry 0 rz 0 deg; joints [32.425, -33.605, 91.822, 37.074, -62.777, -18.243]
  Set speed (1000.0 mm/s)
  MoveL 220 to (-219.16, 498.42, 5) mm, rotated rx -180 ry 0 rz 0 deg; joints [32.421, -34.033, 91.915, 37.175, -62.509, -18.469]
  MoveL 221 to (-219.16, 499.69, 5) mm, rotated rx -180 ry 0 rz 0 deg; joints [32.459, -34.003, 91.845, 37.228, -62.489, -18.514]
  Set speed (25.4 mm/s)
  MoveL 222 to (-219.16, 499.69, 1.82) mm, rotated rx -180 ry 0 rz 0 deg; joints [32.46, -33.844, 91.811, 37.19, -62.589, -18.429]
  MoveL 223 to (-219.16, 499.69, -7.72) mm, rotated rx 180 ry 0 rz 0 deg; joints [32.465, -33.364, 91.705, 37.078, -62.888, -18.178]
  MoveC 224 to (-218.98, 499.69, -8.16) mm, rotated rx 180 ry 0 rz 0 deg; joints [32.468, -33.349, 91.716, 37.074, -62.91, -18.162] to (-218.53, 499.69, -8.35) mm, rotated rx 180 ry 0 rz 0 deg; joints [32.477, -33.357, 91.753, 37.074, -62.936, -18.147]
  Set speed (50.8 mm/s)
  MoveL 225 to (-217.89, 499.69, -8.35) mm, rotated rx -180 ry 0 rz 0 deg; joints [32.489, -33.382, 91.808, 37.078, -62.964, -18.131]
  MoveC 226 to (-217.44, 499.51, -8.35) mm, rotated rx -180 ry 0 rz 0 deg; joints [32.492, -33.404, 91.858, 37.073, -62.987, -18.114] to (-217.26, 499.06, -8.35) mm, rotated rx -180 ry 0 rz 0 deg; joints [32.482, -33.422, 91.899, 37.055, -63.002, -18.094]
  MoveL 227 to (-217.26, 473.66, -8.35) mm, rotated rx -180 ry 0 rz 0 deg; joints [31.714, -34.019, 93.28, 36.001, -63.396, -17.214]
  MoveL 228 to (-268.06, 473.66, -8.35) mm, rotated rx -180 ry 0 rz 0 deg; joints [30.782, -31.996, 88.749, 35.774, -61.074, -18.423]
  MoveL 229 to (-268.06, 524.46, -8.35) mm, rotated rx 180 ry 0 rz 0 deg; joints [32.281, -30.731, 85.874, 37.935, -60.29, -20.3]
  MoveL 230 to (-217.26, 524.46, -8.35) mm, rotated rx -180 ry 0 rz 0 deg; joints [33.237, -32.799, 90.468, 38.112, -62.605, -19.004]
  MoveL 231 to (-217.26, 499.06, -8.35) mm, rotated rx -180 ry 0 rz 0 deg; joints [32.482, -33.422, 91.899, 37.055, -63.002, -18.094]
  MoveC 232 to (-217.44, 498.61, -8.35) mm, rotated rx -180 ry 0 rz 0 deg; joints [32.465, -33.425, 91.907, 37.035, -63.001, -18.083] to (-217.89, 498.42, -8.35) mm, rotated rx 180 ry 0 rz 0 deg; joints [32.451, -33.412, 91.878, 37.025, -62.984, -18.087]
  MoveL 233 to (-218.53, 498.42, -8.35) mm, rotated rx -180 ry 0 rz 0 deg; joints [32.439, -33.388, 91.823, 37.022, -62.956, -18.102]
  MoveC 234 to (-218.98, 498.42, -8.16) mm, rotated rx -180 ry 0 rz 0 deg; joints [32.43, -33.379, 91.786, 37.021, -62.93, -18.117] to (-219.16, 498.42, -7.72) mm, rotated rx 180 ry 0 rz 0 deg; joints [32.427, -33.395, 91.775, 37.025, -62.908, -18.133]
  Set speed (1000.0 mm/s)
  MoveL 235 to (-219.16, 498.42, 6) mm, rotated rx -180 ry 0 rz 0 deg; joints [32.421, -34.083, 91.926, 37.187, -62.477, -18.496]
  MoveL 236 to (-346.16, 499.69, 6) mm, rotated rx -180 ry 0 rz 0 deg; joints [30.191, -28.578, 79.871, 37.093, -56.474, -21.887]
  Set speed (25.4 mm/s)
  MoveL 237 to (-346.16, 499.69, -3.54) mm, rotated rx -180 ry 0 rz 0 deg; joints [30.195, -28.13, 79.762, 36.962, -56.746, -21.645]
  MoveC 238 to (-345.98, 499.69, -3.99) mm, rotated rx -180 ry 0 rz 0 deg; joints [30.198, -28.118, 79.775, 36.956, -56.768, -21.628] to (-345.53, 499.69, -4.17) mm, rotated rx -180 ry 0 rz 0 deg; joints [30.206, -28.13, 79.819, 36.952, -56.796, -21.61]
  Set speed (50.8 mm/s)
  MoveL 239 to (-344.89, 499.69, -4.17) mm, rotated rx -180 ry 0 rz 0 deg; joints [30.216, -28.16, 79.884, 36.95, -56.828, -21.591]
  MoveC 240 to (-344.44, 499.51, -4.18) mm, rotated rx -180 ry 0 rz 0 deg; joints [30.219, -28.186, 79.941, 36.94, -56.853, -21.571] to (-344.26, 499.06, -4.17) mm, rotated rx -180 ry 0 rz 0 deg; joints [30.209, -28.207, 79.987, 36.919, -56.87, -21.547]
  MoveL 241 to (-344.26, 473.66, -4.18) mm, rotated rx 180 ry 0 rz 0 deg; joints [29.472, -28.87, 81.464, 35.789, -57.257, -20.539]
  MoveL 242 to (-395.06, 473.66, -4.18) mm, rotated rx 180 ry 0 rz 0 deg; joints [28.655, -26.415, 76.131, 36.013, -54.626, -22.074]
  MoveL 243 to (-395.06, 524.46, -4.17) mm, rotated rx -180 ry 0 rz 0 deg; joints [30.093, -24.977, 72.974, 38.387, -53.828, -24.284]
  MoveL 244 to (-344.26, 524.46, -4.17) mm, rotated rx -180 ry 0 rz 0 deg; joints [30.934, -27.513, 78.448, 38.061, -56.475, -22.593]
  MoveL 245 to (-344.26, 499.06, -4.17) mm, rotated rx -180 ry 0 rz 0 deg; joints [30.209, -28.207, 79.987, 36.919, -56.87, -21.547]
  MoveC 246 to (-344.44, 498.61, -4.17) mm, rotated rx -180 ry 0 rz 0 deg; joints [30.193, -28.21, 79.995, 36.9, -56.867, -21.534] to (-344.89, 498.42, -4.17) mm, rotated rx -180 ry 0 rz 0 deg; joints [30.18, -28.194, 79.96, 36.893, -56.847, -21.54]
  MoveL 247 to (-345.53, 498.42, -4.18) mm, rotated rx 180 ry 0 rz 0 deg; joints [30.169, -28.164, 79.895, 36.895, -56.815, -21.559]
  MoveC 248 to (-345.98, 498.42, -3.99) mm, rotated rx 180 ry 0 rz 0 deg; joints [30.162, -28.152, 79.851, 36.899, -56.787, -21.577] to (-346.16, 498.42, -3.54) mm, rotated rx -180 ry 0 rz 0 deg; joints [30.158, -28.164, 79.837, 36.905, -56.765, -21.594]
  Set speed (1000.0 mm/s)
  MoveL 249 to (-346.16, 498.42, 5) mm, rotated rx 180 ry 0 rz 0 deg; joints [30.155, -28.566, 79.935, 37.022, -56.522, -21.81]
  MoveL 250 to (-346.16, 499.69, 5) mm, rotated rx -180 ry 0 rz 0 deg; joints [30.192, -28.531, 79.86, 37.079, -56.502, -21.862]
  Set speed (25.4 mm/s)
  MoveL 251 to (-346.16, 499.69, 1.83) mm, rotated rx -180 ry 0 rz 0 deg; joints [30.193, -28.383, 79.824, 37.035, -56.593, -21.781]
  MoveL 252 to (-346.16, 499.69, -7.72) mm, rotated rx 180 ry 0 rz 0 deg; joints [30.197, -27.933, 79.711, 36.906, -56.864, -21.541]
  MoveC 253 to (-345.98, 499.69, -8.16) mm, rotated rx -180 ry 0 rz 0 deg; joints [30.2, -27.921, 79.725, 36.9, -56.886, -21.524] to (-345.53, 499.69, -8.35) mm, rotated rx 180 ry 0 rz 0 deg; joints [30.207, -27.933, 79.769, 36.896, -56.914, -21.506]
  Set speed (50.8 mm/s)
  MoveL 254 to (-344.89, 499.69, -8.35) mm, rotated rx -180 ry 0 rz 0 deg; joints [30.218, -27.963, 79.834, 36.894, -56.946, -21.487]
  MoveC 255 to (-344.44, 499.51, -8.35) mm, rotated rx 180 ry 0 rz 0 deg; joints [30.22, -27.989, 79.891, 36.884, -56.971, -21.466] to (-344.26, 499.06, -8.35) mm, rotated rx 180 ry 0 rz 0 deg; joints [30.21, -28.01, 79.937, 36.864, -56.988, -21.442]
  MoveL 256 to (-344.26, 473.66, -8.35) mm, rotated rx -180 ry 0 rz 0 deg; joints [29.474, -28.672, 81.414, 35.735, -57.378, -20.436]
  MoveL 257 to (-395.06, 473.66, -8.35) mm, rotated rx -180 ry 0 rz 0 deg; joints [28.657, -26.221, 76.079, 35.955, -54.742, -21.972]
  MoveL 258 to (-395.06, 524.46, -8.35) mm, rotated rx 180 ry 0 rz 0 deg; joints [30.094, -24.785, 72.92, 38.326, -53.938, -24.178]
  MoveL 259 to (-344.26, 524.46, -8.35) mm, rotated rx 180 ry 0 rz 0 deg; joints [30.936, -27.317, 78.397, 38.003, -56.59, -22.486]
  MoveL 260 to (-344.26, 499.06, -8.35) mm, rotated rx 180 ry 0 rz 0 deg; joints [30.21, -28.01, 79.937, 36.864, -56.988, -21.442]
  MoveC 261 to (-344.44, 498.61, -8.35) mm, rotated rx -180 ry 0 rz 0 deg; joints [30.194, -28.013, 79.944, 36.844, -56.985, -21.43] to (-344.89, 498.42, -8.35) mm, rotated rx -180 ry 0 rz 0 deg; joints [30.182, -27.997, 79.909, 36.837, -56.965, -21.436]
  MoveL 262 to (-345.53, 498.42, -8.35) mm, rotated rx -180 ry 0 rz 0 deg; joints [30.171, -27.967, 79.844, 36.839, -56.933, -21.455]
  MoveC 263 to (-345.98, 498.42, -8.16) mm, rotated rx 180 ry 0 rz 0 deg; joints [30.163, -27.955, 79.801, 36.843, -56.905, -21.473] to (-346.16, 498.42, -7.72) mm, rotated rx -180 ry 0 rz 0 deg; joints [30.16, -27.967, 79.787, 36.849, -56.883, -21.489]
  Set speed (1000.0 mm/s)
  MoveL 264 to (-346.16, 498.42, 6) mm, rotated rx -180 ry 0 rz 0 deg; joints [30.155, -28.612, 79.946, 37.035, -56.493, -21.836]
  MoveL 265 to (139.15, 499.69, 6) mm, rotated rx -180 ry 0 rz 0 deg; joints [40.798, -45.472, 118.387, 42.253, -76.297, -11.122]
  Set speed (25.4 mm/s)
  MoveL 266 to (139.15, 499.69, -3.54) mm, rotated rx 180 ry 0 rz 0 deg; joints [40.804, -44.87, 118.28, 42.179, -76.664, -10.782]
  MoveC 267 to (139.34, 499.69, -3.99) mm, rotated rx -180 ry 0 rz 0 deg; joints [40.809, -44.847, 118.287, 42.18, -76.687, -10.762] to (139.79, 499.69, -4.17) mm, rotated rx 180 ry 0 rz 0 deg; joints [40.822, -44.846, 118.313, 42.188, -76.71, -10.747]
  Set speed (50.8 mm/s)
  MoveL 268 to (140.42, 499.69, -4.18) mm, rotated rx 180 ry 0 rz 0 deg; joints [40.84, -44.862, 118.353, 42.203, -76.731, -10.734]
  MoveC 269 to (140.87, 499.51, -4.17) mm, rotated rx 180 ry 0 rz 0 deg; joints [40.847, -44.877, 118.391, 42.205, -76.75, -10.719] to (141.06, 499.06, -4.18) mm, rotated rx -180 ry 0 rz 0 deg; joints [40.837, -44.891, 118.427, 42.192, -76.764, -10.702]
  MoveL 270 to (141.06, 473.66, -4.17) mm, rotated rx -180 ry 0 rz 0 deg; joints [39.995, -45.399, 119.788, 41.212, -77.246, -9.942]
  MoveL 271 to (90.26, 473.66, -4.18) mm, rotated rx -180 ry 0 rz 0 deg; joints [38.606, -44.101, 116.507, 40.121, -75.484, -10.961]
  MoveL 272 to (90.26, 524.46, -4.18) mm, rotated rx 180 ry 0 rz 0 deg; joints [40.256, -43.042, 113.77, 42.087, -74.562, -12.51]
  MoveL 273 to (141.06, 524.46, -4.18) mm, rotated rx 180 ry 0 rz 0 deg; joints [41.659, -44.362, 117.032, 43.161, -76.289, -11.486]
  MoveL 274 to (141.06, 499.06, -4.18) mm, rotated rx -180 ry 0 rz 0 deg; joints [40.837, -44.891, 118.427, 42.192, -76.764, -10.702]
  MoveC 275 to (140.87, 498.61, -4.17) mm, rotated rx 180 ry 0 rz 0 deg; joints [40.817, -44.895, 118.44, 42.171, -76.767, -10.692] to (140.42, 498.42, -4.17) mm, rotated rx -180 ry 0 rz 0 deg; joints [40.798, -44.888, 118.422, 42.154, -76.755, -10.695]
  MoveL 276 to (139.79, 498.42, -4.18) mm, rotated rx -180 ry 0 rz 0 deg; joints [40.78, -44.872, 118.382, 42.139, -76.734, -10.708]
  MoveC 277 to (139.34, 498.42, -3.99) mm, rotated rx -180 ry 0 rz 0 deg; joints [40.768, -44.873, 118.356, 42.131, -76.711, -10.724] to (139.15, 498.42, -3.54) mm, rotated rx -180 ry 0 rz 0 deg; joints [40.762, -44.896, 118.349, 42.13, -76.688, -10.743]
  Set speed (1000.0 mm/s)
  MoveL 278 to (139.15, 498.42, 5) mm, rotated rx -180 ry 0 rz 0 deg; joints [40.757, -45.436, 118.446, 42.196, -76.359, -11.048]
  MoveL 279 to (139.15, 499.69, 5) mm, rotated rx -180 ry 0 rz 0 deg; joints [40.799, -45.409, 118.377, 42.245, -76.335, -11.086]
  Set speed (25.4 mm/s)
  MoveL 280 to (139.15, 499.69, 1.83) mm, rotated rx -180 ry 0 rz 0 deg; joints [40.801, -45.209, 118.342, 42.22, -76.458, -10.973]
  MoveL 281 to (139.15, 499.69, -7.72) mm, rotated rx -180 ry 0 rz 0 deg; joints [40.806, -44.607, 118.231, 42.147, -76.824, -10.634]
  MoveC 282 to (139.34, 499.69, -8.16) mm, rotated rx 180 ry 0 rz 0 deg; joints [40.812, -44.583, 118.237, 42.148, -76.847, -10.615] to (139.79, 499.69, -8.35) mm, rotated rx -180 ry 0 rz 0 deg; joints [40.825, -44.582, 118.263, 42.157, -76.869, -10.599]
  Set speed (50.8 mm/s)
  MoveL 283 to (140.42, 499.69, -8.35) mm, rotated rx -180 ry 0 rz 0 deg; joints [40.842, -44.598, 118.303, 42.171, -76.891, -10.586]
  MoveC 284 to (140.87, 499.51, -8.35) mm, rotated rx -180 ry 0 rz 0 deg; joints [40.849, -44.613, 118.342, 42.174, -76.909, -10.571] to (141.06, 499.06, -8.35) mm, rotated rx -180 ry 0 rz 0 deg; joints [40.84, -44.626, 118.378, 42.161, -76.924, -10.554]
  MoveL 285 to (141.06, 473.66, -8.35) mm, rotated rx -180 ry 0 rz 0 deg; joints [39.997, -45.131, 119.738, 41.182, -77.41, -9.795]
  MoveL 286 to (90.26, 473.66, -8.35) mm, rotated rx -180 ry 0 rz 0 deg; joints [38.608, -43.842, 116.458, 40.088, -75.645, -10.822]
  MoveL 287 to (90.26, 524.46, -8.35) mm, rotated rx -180 ry 0 rz 0 deg; joints [40.258, -42.79, 113.722, 42.051, -74.713, -12.369]
  MoveL 288 to (141.06, 524.46, -8.35) mm, rotated rx -180 ry 0 rz 0 deg; joints [41.661, -44.102, 116.982, 43.129, -76.443, -11.338]
  MoveL 289 to (141.06, 499.06, -8.35) mm, rotated rx -180 ry 0 rz 0 deg; joints [40.84, -44.626, 118.378, 42.161, -76.924, -10.554]
  MoveC 290 to (140.87, 498.61, -8.35) mm, rotated rx 180 ry 0 rz 0 deg; joints [40.82, -44.631, 118.39, 42.14, -76.926, -10.544] to (140.42, 498.42, -8.35) mm, rotated rx 180 ry 0 rz 0 deg; joints [40.801, -44.624, 118.372, 42.123, -76.915, -10.548]
  MoveL 291 to (139.79, 498.42, -8.35) mm, rotated rx -180 ry 0 rz 0 deg; joints [40.783, -44.608, 118.332, 42.108, -76.893, -10.56]
  MoveC 292 to (139.34, 498.42, -8.16) mm, rotated rx -180 ry 0 rz 0 deg; joints [40.77, -44.608, 118.306, 42.099, -76.871, -10.576] to (139.15, 498.42, -7.72) mm, rotated rx 180 ry 0 rz 0 deg; joints [40.765, -44.632, 118.3, 42.099, -76.848, -10.596]
  Set speed (1000.0 mm/s)
  MoveL 293 to (139.15, 498.42, 6) mm, rotated rx -180 ry 0 rz 0 deg; joints [40.757, -45.499, 118.456, 42.204, -76.32, -11.084]
  MoveL 294 to (266.15, 499.69, 6) mm, rotated rx 180 ry 0 rz 0 deg; joints [44.659, -48.449, 125.994, 45.472, -80.316, -8.573]
  Set speed (25.4 mm/s)
  MoveL 295 to (266.15, 499.69, -3.54) mm, rotated rx -180 ry 0 rz 0 deg; joints [44.665, -47.789, 125.881, 45.413, -80.7, -8.179]
  MoveC 296 to (266.34, 499.69, -3.99) mm, rotated rx -180 ry 0 rz 0 deg; joints [44.671, -47.762, 125.886, 45.416, -80.724, -8.157] to (266.79, 499.69, -4.17) mm, rotated rx -180 ry 0 rz 0 deg; joints [44.686, -47.759, 125.909, 45.428, -80.745, -8.14]
  Set speed (50.8 mm/s)
  MoveL 297 to (267.42, 499.69, -4.17) mm, rotated rx -180 ry 0 rz 0 deg; joints [44.707, -47.772, 125.945, 45.446, -80.764, -8.127]
  MoveC 298 to (267.87, 499.51, -4.17) mm, rotated rx 180 ry 0 rz 0 deg; joints [44.716, -47.785, 125.981, 45.452, -80.781, -8.111] to (268.06, 499.06, -4.17) mm, rotated rx -180 ry 0 rz 0 deg; joints [44.707, -47.797, 126.017, 45.44, -80.796, -8.093]
  MoveL 299 to (268.06, 473.66, -4.17) mm, rotated rx 180 ry 0 rz 0 deg; joints [43.854, -48.276, 127.415, 44.483, -81.328, -7.315]
  MoveL 300 to (217.26, 473.66, -4.17) mm, rotated rx -180 ry 0 rz 0 deg; joints [42.24, -47.188, 124.461, 43.079, -79.753, -8.383]
  MoveL 301 to (217.26, 524.46, -4.17) mm, rotated rx -180 ry 0 rz 0 deg; joints [43.918, -46.185, 121.664, 45, -78.739, -9.941]
  MoveL 302 to (268.06, 524.46, -4.17) mm, rotated rx -180 ry 0 rz 0 deg; joints [45.535, -47.297, 124.585, 46.382, -80.274, -8.895]
  MoveL 303 to (268.06, 499.06, -4.17) mm, rotated rx -180 ry 0 rz 0 deg; joints [44.707, -47.797, 126.017, 45.44, -80.796, -8.093]
  MoveC 304 to (267.87, 498.61, -4.18) mm, rotated rx -180 ry 0 rz 0 deg; joints [44.686, -47.802, 126.031, 45.418, -80.799, -8.083] to (267.42, 498.42, -4.17) mm, rotated rx 180 ry 0 rz 0 deg; joints [44.665, -47.796, 126.016, 45.398, -80.79, -8.087]
  MoveL 305 to (266.79, 498.42, -4.18) mm, rotated rx -180 ry 0 rz 0 deg; joints [44.644, -47.783, 125.98, 45.38, -80.771, -8.1]
  MoveC 306 to (266.34, 498.42, -3.99) mm, rotated rx 180 ry 0 rz 0 deg; joints [44.629, -47.787, 125.957, 45.368, -80.75, -8.117] to (266.15, 498.42, -3.54) mm, rotated rx -180 ry 0 rz 0 deg; joints [44.623, -47.814, 125.952, 45.366, -80.726, -8.14]
  Set speed (1000.0 mm/s)
  MoveL 307 to (266.15, 498.42, 5) mm, rotated rx -180 ry 0 rz 0 deg; joints [44.617, -48.405, 126.053, 45.418, -80.382, -8.492]
  MoveL 308 to (266.15, 499.69, 5) mm, rotated rx -180 ry 0 rz 0 deg; joints [44.659, -48.38, 125.983, 45.466, -80.356, -8.532]
  Set speed (25.4 mm/s)
  MoveL 309 to (266.15, 499.69, 1.83) mm, rotated rx 180 ry 0 rz 0 deg; joints [44.662, -48.161, 125.946, 45.446, -80.484, -8.4]
  MoveL 310 to (266.15, 499.69, -7.71) mm, rotated rx -180 ry 0 rz 0 deg; joints [44.668, -47.5, 125.829, 45.389, -80.867, -8.008]
  MoveC 311 to (266.34, 499.69, -8.16) mm, rotated rx 180 ry 0 rz 0 deg; joints [44.674, -47.473, 125.834, 45.391, -80.891, -7.986] to (266.79, 499.69, -8.35) mm, rotated rx -180 ry 0 rz 0 deg; joints [44.689, -47.469, 125.857, 45.403, -80.912, -7.969]
  Set speed (50.8 mm/s)
  MoveL 312 to (267.42, 499.69, -8.35) mm, rotated rx -180 ry 0 rz 0 deg; joints [44.71, -47.482, 125.893, 45.421, -80.931, -7.956]
  MoveC 313 to (267.87, 499.51, -8.35) mm, rotated rx -180 ry 0 rz 0 deg; joints [44.718, -47.495, 125.929, 45.427, -80.948, -7.94] to (268.06, 499.06, -8.35) mm, rotated rx -180 ry 0 rz 0 deg; joints [44.709, -47.507, 125.964, 45.416, -80.963, -7.922]
  MoveL 314 to (268.06, 473.66, -8.35) mm, rotated rx 180 ry 0 rz 0 deg; joints [43.857, -47.981, 127.362, 44.46, -81.502, -7.144]
  MoveL 315 to (217.26, 473.66, -8.35) mm, rotated rx -180 ry 0 rz 0 deg; joints [42.243, -46.904, 124.409, 43.053, -79.923, -8.222]
  MoveL 316 to (217.26, 524.46, -8.35) mm, rotated rx 180 ry 0 rz 0 deg; joints [43.921, -45.91, 121.614, 44.972, -78.897, -9.78]
  MoveL 317 to (268.06, 524.46, -8.35) mm, rotated rx -180 ry 0 rz 0 deg; joints [45.538, -47.013, 124.534, 46.356, -80.435, -8.725]
  MoveL 318 to (268.06, 499.06, -8.35) mm, rotated rx -180 ry 0 rz 0 deg; joints [44.709, -47.507, 125.964, 45.416, -80.963, -7.922]
  MoveC 319 to (267.87, 498.61, -8.35) mm, rotated rx -180 ry 0 rz 0 deg; joints [44.689, -47.512, 125.979, 45.394, -80.967, -7.912] to (267.42, 498.42, -8.35) mm, rotated rx 180 ry 0 rz 0 deg; joints [44.668, -47.506, 125.964, 45.374, -80.957, -7.916]
  MoveL 320 to (266.79, 498.42, -8.35) mm, rotated rx -180 ry 0 rz 0 deg; joints [44.647, -47.493, 125.928, 45.356, -80.938, -7.929]
  MoveC 321 to (266.34, 498.42, -8.16) mm, rotated rx -180 ry 0 rz 0 deg; joints [44.632, -47.497, 125.905, 45.344, -80.917, -7.947] to (266.15, 498.42, -7.72) mm, rotated rx -180 ry 0 rz 0 deg; joints [44.626, -47.524, 125.9, 45.341, -80.894, -7.969]
  Set speed (1000.0 mm/s)
  MoveL 322 to (266.15, 498.42, 6) mm, rotated rx -180 ry 0 rz 0 deg; joints [44.617, -48.474, 126.065, 45.425, -80.341, -8.534]
  MoveL 323 to (393.15, 499.69, 6) mm, rotated rx -180 ry 0 rz 0 deg; joints [49.128, -50.922, 132.788, 49.504, -83.823, -5.905]
  Set speed (25.4 mm/s)
  MoveL 324 to (393.15, 499.69, -3.54) mm, rotated rx -180 ry 0 rz 0 deg; joints [49.135, -50.196, 132.668, 49.463, -84.217, -5.443]
  MoveC 325 to (393.34, 499.69, -3.99) mm, rotated rx -180 ry 0 rz 0 deg; joints [49.142, -50.165, 132.671, 49.468, -84.24, -5.417] to (393.79, 499.69, -4.17) mm, rotated rx -180 ry 0 rz 0 deg; joints [49.159, -50.159, 132.691, 49.483, -84.259, -5.398]
  Set speed (50.8 mm/s)
  MoveL 326 to (394.42, 499.69, -4.17) mm, rotated rx -180 ry 0 rz 0 deg; joints [49.183, -50.169, 132.723, 49.505, -84.275, -5.384]
  MoveC 327 to (394.87, 499.51, -4.17) mm, rotated rx -180 ry 0 rz 0 deg; joints [49.194, -50.18, 132.756, 49.514, -84.291, -5.368] to (395.06, 499.06, -4.17) mm, rotated rx -180 ry 0 rz 0 deg; joints [49.187, -50.191, 132.792, 49.505, -84.306, -5.349]
  MoveL 328 to (395.06, 473.66, -4.17) mm, rotated rx -180 ry 0 rz 0 deg; joints [48.341, -50.631, 134.244, 48.586, -84.892, -4.514]
  MoveL 329 to (344.26, 473.66, -4.17) mm, rotated rx -180 ry 0 rz 0 deg; joints [46.464, -49.752, 131.608, 46.84, -83.535, -5.659]
  MoveL 330 to (344.26, 524.46, -4.17) mm, rotated rx -180 ry 0 rz 0 deg; joints [48.141, -48.815, 128.719, 48.696, -82.42, -7.295]
  MoveL 331 to (395.06, 524.46, -4.18) mm, rotated rx 180 ry 0 rz 0 deg; joints [50.005, -49.727, 131.31, 50.404, -83.737, -6.205]
  MoveL 332 to (395.06, 499.06, -4.17) mm, rotated rx -180 ry 0 rz 0 deg; joints [49.187, -50.191, 132.792, 49.505, -84.306, -5.349]
  MoveC 333 to (394.87, 498.61, -4.17) mm, rotated rx -180 ry 0 rz 0 deg; joints [49.165, -50.196, 132.808, 49.482, -84.311, -5.338] to (394.42, 498.42, -4.17) mm, rotated rx -180 ry 0 rz 0 deg; joints [49.142, -50.192, 132.796, 49.46, -84.304, -5.342]
  MoveL 334 to (393.79, 498.42, -4.18) mm, rotated rx -180 ry 0 rz 0 deg; joints [49.118, -50.181, 132.765, 49.437, -84.288, -5.356]
  MoveC 335 to (393.34, 498.42, -3.99) mm, rotated rx 180 ry 0 rz 0 deg; joints [49.101, -50.188, 132.744, 49.422, -84.269, -5.375] to (393.15, 498.42, -3.54) mm, rotated rx -180 ry 0 rz 0 deg; joints [49.093, -50.219, 132.741, 49.417, -84.245, -5.401]
  Set speed (1000.0 mm/s)
  MoveL 336 to (393.15, 498.42, 5) mm, rotated rx 180 ry 0 rz 0 deg; joints [49.087, -50.869, 132.849, 49.454, -83.892, -5.814]
  MoveL 337 to (393.15, 499.69, 5) mm, rotated rx -180 ry 0 rz 0 deg; joints [49.129, -50.846, 132.776, 49.5, -83.864, -5.856]
  Set speed (25.4 mm/s)
  MoveL 338 to (393.15, 499.69, 1.82) mm, rotated rx 180 ry 0 rz 0 deg; joints [49.131, -50.605, 132.736, 49.486, -83.996, -5.702]
  MoveL 339 to (393.15, 499.69, -7.71) mm, rotated rx -180 ry 0 rz 0 deg; joints [49.138, -49.878, 132.612, 49.446, -84.388, -5.243]
  MoveC 340 to (393.34, 499.69, -8.16) mm, rotated rx -180 ry 0 rz 0 deg; joints [49.145, -49.847, 132.616, 49.451, -84.411, -5.217] to (393.79, 499.69, -8.35) mm, rotated rx -180 ry 0 rz 0 deg; joints [49.162, -49.84, 132.636, 49.466, -84.43, -5.198]
  Set speed (50.8 mm/s)
  MoveL 341 to (394.42, 499.69, -8.35) mm, rotated rx -180 ry 0 rz 0 deg; joints [49.186, -49.851, 132.667, 49.488, -84.446, -5.184]
  MoveC 342 to (394.87, 499.51, -8.35) mm, rotated rx -180 ry 0 rz 0 deg; joints [49.197, -49.862, 132.701, 49.498, -84.462, -5.167] to (395.06, 499.06, -8.35) mm, rotated rx -180 ry 0 rz 0 deg; joints [49.19, -49.873, 132.736, 49.488, -84.477, -5.148]
  MoveL 343 to (395.06, 473.66, -8.35) mm, rotated rx 180 ry 0 rz 0 deg; joints [48.344, -50.306, 134.187, 48.572, -85.071, -4.312]
  MoveL 344 to (344.26, 473.66, -8.35) mm, rotated rx 180 ry 0 rz 0 deg; joints [46.467, -49.438, 131.553, 46.822, -83.712, -5.47]
  MoveL 345 to (344.26, 524.46, -8.35) mm, rotated rx -180 ry 0 rz 0 deg; joints [48.143, -48.514, 128.666, 48.674, -82.583, -7.109]
  MoveL 346 to (395.06, 524.46, -8.35) mm, rotated rx -180 ry 0 rz 0 deg; joints [50.008, -49.415, 131.255, 50.386, -83.901, -6.006]
  MoveL 347 to (395.06, 499.06, -8.35) mm, rotated rx -180 ry 0 rz 0 deg; joints [49.19, -49.873, 132.736, 49.488, -84.477, -5.148]
  MoveC 348 to (394.87, 498.61, -8.35) mm, rotated rx -180 ry 0 rz 0 deg; joints [49.168, -49.877, 132.753, 49.466, -84.482, -5.137] to (394.42, 498.42, -8.35) mm, rotated rx -180 ry 0 rz 0 deg; joints [49.145, -49.873, 132.741, 49.443, -84.475, -5.141]
  MoveL 349 to (393.79, 498.42, -8.35) mm, rotated rx -180 ry 0 rz 0 deg; joints [49.121, -49.863, 132.709, 49.421, -84.459, -5.156]
  MoveC 350 to (393.34, 498.42, -8.16) mm, rotated rx 180 ry 0 rz 0 deg; joints [49.104, -49.869, 132.689, 49.405, -84.44, -5.175] to (393.15, 498.42, -7.72) mm, rotated rx 180 ry 0 rz 0 deg; joints [49.096, -49.901, 132.686, 49.401, -84.417, -5.2]
  Set speed (1000.0 mm/s)
  MoveL 351 to (393.15, 498.42, 6) mm, rotated rx -180 ry 0 rz 0 deg; joints [49.086, -50.946, 132.861, 49.458, -83.851, -5.863]
  MoveL 352 to (393.15, 313.35, 6) mm, rotated rx -180 ry 0 rz 0 deg; joints [42.207, -53.714, 142.748, 42.216, -88.415, -0.377]
  Set speed (25.4 mm/s)
  MoveL 353 to (393.15, 313.35, -3.54) mm, rotated rx -180 ry 0 rz 0 deg; joints [42.214, -52.856, 142.609, 42.213, -88.948, 0.106]
  MoveC 354 to (393.34, 313.35, -3.99) mm, rotated rx -180 ry 0 rz 0 deg; joints [42.221, -52.818, 142.613, 42.22, -88.978, 0.134] to (393.79, 313.36, -4.17) mm, rotated rx -180 ry 0 rz 0 deg; joints [42.239, -52.808, 142.634, 42.236, -89.002, 0.156]
  Set speed (50.8 mm/s)
  MoveL 355 to (394.42, 313.35, -4.17) mm, rotated rx -180 ry 0 rz 0 deg; joints [42.263, -52.816, 142.668, 42.26, -89.021, 0.173]
  MoveC 356 to (394.87, 313.17, -4.17) mm, rotated rx -180 ry 0 rz 0 deg; joints [42.272, -52.824, 142.702, 42.269, -89.04, 0.19] to (395.06, 312.72, -4.18) mm, rotated rx 180 ry 0 rz 0 deg; joints [42.26, -52.831, 142.734, 42.257, -89.058, 0.207]
  MoveL 357 to (395.06, 287.32, -4.18) mm, rotated rx 180 ry 0 rz 0 deg; joints [41.176, -53.082, 143.957, 41.166, -89.789, 0.848]
  MoveL 358 to (344.26, 287.32, -4.17) mm, rotated rx -180 ry 0 rz 0 deg; joints [39.319, -52.384, 141.124, 39.333, -88.156, -0.526]
  MoveL 359 to (344.26, 338.12, -4.17) mm, rotated rx 180 ry 0 rz 0 deg; joints [41.434, -51.793, 138.703, 41.502, -86.814, -1.775]
  MoveL 360 to (395.06, 338.12, -4.18) mm, rotated rx -180 ry 0 rz 0 deg; joints [43.309, -52.553, 141.478, 43.321, -88.348, -0.466]
  MoveL 361 to (395.06, 312.72, -4.18) mm, rotated rx 180 ry 0 rz 0 deg; joints [42.26, -52.831, 142.734, 42.257, -89.058, 0.207]
  MoveC 362 to (394.87, 312.27, -4.17) mm, rotated rx -180 ry 0 rz 0 deg; joints [42.234, -52.833, 142.746, 42.231, -89.065, 0.213] to (394.42, 312.08, -4.17) mm, rotated rx 180 ry 0 rz 0 deg; joints [42.21, -52.829, 142.73, 42.206, -89.057, 0.206]
  MoveL 363 to (393.79, 312.08, -4.18) mm, rotated rx -180 ry 0 rz 0 deg; joints [42.185, -52.821, 142.696, 42.183, -89.038, 0.189]
  MoveC 364 to (393.34, 312.09, -3.99) mm, rotated rx 180 ry 0 rz 0 deg; joints [42.168, -52.832, 142.675, 42.166, -89.014, 0.167] to (393.15, 312.08, -3.54) mm, rotated rx 180 ry 0 rz 0 deg; joints [42.161, -52.87, 142.671, 42.159, -88.983, 0.139]
  Set speed (1000.0 mm/s)
  MoveL 365 to (393.15, 312.08, 5) mm, rotated rx -180 ry 0 rz 0 deg; joints [42.154, -53.638, 142.796, 42.162, -88.506, -0.293]
  MoveL 366 to (393.15, 313.36, 5) mm, rotated rx -180 ry 0 rz 0 deg; joints [42.207, -53.624, 142.734, 42.216, -88.471, -0.326]
  Set speed (25.4 mm/s)
  MoveL 367 to (393.15, 313.36, 1.82) mm, rotated rx 180 ry 0 rz 0 deg; joints [42.21, -53.339, 142.688, 42.214, -88.649, -0.165]
  MoveL 368 to (393.15, 313.35, -7.71) mm, rotated rx -180 ry 0 rz 0 deg; joints [42.217, -52.481, 142.546, 42.212, -89.179, 0.316]
  MoveC 369 to (393.34, 313.36, -8.16) mm, rotated rx -180 ry 0 rz 0 deg; joints [42.225, -52.443, 142.549, 42.219, -89.209, 0.344] to (393.79, 313.36, -8.35) mm, rotated rx -180 ry 0 rz 0 deg; joints [42.242, -52.432, 142.57, 42.236, -89.233, 0.365]
  Set speed (50.8 mm/s)
  MoveL 370 to (394.42, 313.36, -8.35) mm, rotated rx 180 ry 0 rz 0 deg; joints [42.266, -52.44, 142.605, 42.26, -89.252, 0.383]
  MoveC 371 to (394.87, 313.17, -8.35) mm, rotated rx 180 ry 0 rz 0 deg; joints [42.275, -52.448, 142.638, 42.269, -89.271, 0.4] to (395.06, 312.72, -8.35) mm, rotated rx -180 ry 0 rz 0 deg; joints [42.264, -52.455, 142.67, 42.258, -89.29, 0.417]
  MoveL 372 to (395.06, 287.32, -8.35) mm, rotated rx 180 ry 0 rz 0 deg; joints [41.179, -52.697, 143.892, 41.169, -90.03, 1.059]
  MoveL 373 to (344.26, 287.32, -8.35) mm, rotated rx -180 ry 0 rz 0 deg; joints [39.322, -52.018, 141.061, 39.331, -88.39, -0.334]
  MoveL 374 to (344.26, 338.12, -8.35) mm, rotated rx 180 ry 0 rz 0 deg; joints [41.437, -51.443, 138.643, 41.495, -87.032, -1.583]
  MoveL 375 to (395.06, 338.12, -8.35) mm, rotated rx -180 ry 0 rz 0 deg; joints [43.312, -52.185, 141.415, 43.319, -88.57, -0.256]
  MoveL 376 to (395.06, 312.72, -8.35) mm, rotated rx -180 ry 0 rz 0 deg; joints [42.264, -52.455, 142.67, 42.258, -89.29, 0.417]
  MoveC 377 to (394.87, 312.27, -8.35) mm, rotated rx -180 ry 0 rz 0 deg; joints [42.238, -52.457, 142.682, 42.231, -89.297, 0.423] to (394.42, 312.09, -8.35) mm, rotated rx -180 ry 0 rz 0 deg; joints [42.213, -52.453, 142.666, 42.207, -89.289, 0.416]
  MoveL 378 to (393.79, 312.09, -8.35) mm, rotated rx 180 ry 0 rz 0 deg; joints [42.189, -52.445, 142.632, 42.183, -89.269, 0.398]
  MoveC 379 to (393.34, 312.09, -8.16) mm, rotated rx -180 ry 0 rz 0 deg; joints [42.171, -52.456, 142.611, 42.166, -89.245, 0.376] to (393.15, 312.08, -7.72) mm, rotated rx -180 ry 0 rz 0 deg; joints [42.164, -52.494, 142.608, 42.159, -89.215, 0.349]
  Set speed (1000.0 mm/s)
  MoveL 380 to (393.15, 312.09, 6) mm, rotated rx 180 ry 0 rz 0 deg; joints [42.153, -53.728, 142.81, 42.162, -88.449, -0.344]
  MoveL 381 to (266.15, 313.35, 6) mm, rotated rx -180 ry 0 rz 0 deg; joints [37.796, -51.571, 135.501, 38.005, -84.339, -3.461]
  Set speed (25.4 mm/s)
  MoveL 382 to (266.15, 313.35, -3.54) mm, rotated rx -180 ry 0 rz 0 deg; joints [37.802, -50.813, 135.376, 37.974, -84.838, -3.071]
  MoveC 383 to (266.34, 313.35, -3.99) mm, rotated rx -180 ry 0 rz 0 deg; joints [37.809, -50.781, 135.381, 37.978, -84.868, -3.048] to (266.79, 313.35, -4.17) mm, rotated rx -180 ry 0 rz 0 deg; joints [37.823, -50.775, 135.405, 37.991, -84.893, -3.03]
  Set speed (50.8 mm/s)
  MoveL 384 to (267.42, 313.35, -4.17) mm, rotated rx -180 ry 0 rz 0 deg; joints [37.843, -50.787, 135.443, 38.01, -84.914, -3.016]
  MoveC 385 to (267.87, 313.17, -4.18) mm, rotated rx -180 ry 0 rz 0 deg; joints [37.85, -50.797, 135.479, 38.015, -84.934, -3.001] to (268.06, 312.72, -4.18) mm, rotated rx -180 ry 0 rz 0 deg; joints [37.837, -50.807, 135.51, 38.001, -84.951, -2.986]
  MoveL 386 to (268.06, 287.32, -4.17) mm, rotated rx -180 ry 0 rz 0 deg; joints [36.785, -51.127, 136.664, 36.905, -85.558, -2.406]
  MoveL 387 to (217.26, 287.32, -4.18) mm, rotated rx -180 ry 0 rz 0 deg; joints [35.246, -50.158, 133.554, 35.48, -83.743, -3.556]
  MoveL 388 to (217.26, 338.12, -4.18) mm, rotated rx 180 ry 0 rz 0 deg; joints [37.291, -49.458, 131.258, 37.647, -82.618, -4.726]
  MoveL 389 to (268.06, 338.12, -4.18) mm, rotated rx -180 ry 0 rz 0 deg; joints [38.861, -50.465, 134.322, 39.077, -84.353, -3.596]
  MoveL 390 to (268.06, 312.72, -4.18) mm, rotated rx -180 ry 0 rz 0 deg; joints [37.837, -50.807, 135.51, 38.001, -84.951, -2.986]
  MoveC 391 to (267.87, 312.27, -4.17) mm, rotated rx 180 ry 0 rz 0 deg; joints [37.813, -50.809, 135.52, 37.977, -84.955, -2.98] to (267.42, 312.09, -4.18) mm, rotated rx -180 ry 0 rz 0 deg; joints [37.791, -50.803, 135.502, 37.956, -84.944, -2.986]
  MoveL 392 to (266.79, 312.09, -4.17) mm, rotated rx -180 ry 0 rz 0 deg; joints [37.771, -50.791, 135.464, 37.937, -84.923, -3]
  MoveC 393 to (266.34, 312.08, -3.99) mm, rotated rx -180 ry 0 rz 0 deg; joints [37.757, -50.798, 135.44, 37.924, -84.898, -3.018] to (266.15, 312.08, -3.54) mm, rotated rx -180 ry 0 rz 0 deg; joints [37.75, -50.83, 135.435, 37.92, -84.868, -3.041]
  Set speed (1000.0 mm/s)
  MoveL 394 to (266.15, 312.08, 5) mm, rotated rx 180 ry 0 rz 0 deg; joints [37.745, -51.509, 135.547, 37.947, -84.421, -3.39]
  MoveL 395 to (266.15, 313.35, 5) mm, rotated rx -180 ry 0 rz 0 deg; joints [37.797, -51.491, 135.488, 38.001, -84.392, -3.42]
  Set speed (25.4 mm/s)
  MoveL 396 to (266.15, 313.36, 1.82) mm, rotated rx -180 ry 0 rz 0 deg; joints [37.799, -51.239, 135.447, 37.991, -84.558, -3.289]
  MoveL 397 to (266.15, 313.35, -7.71) mm, rotated rx 180 ry 0 rz 0 deg; joints [37.805, -50.482, 135.318, 37.962, -85.054, -2.901]
  MoveC 398 to (266.34, 313.36, -8.16) mm, rotated rx 180 ry 0 rz 0 deg; joints [37.811, -50.449, 135.323, 37.966, -85.084, -2.879] to (266.79, 313.36, -8.35) mm, rotated rx -180 ry 0 rz 0 deg; joints [37.826, -50.443, 135.347, 37.979, -85.109, -2.861]
  Set speed (50.8 mm/s)
  MoveL 399 to (267.42, 313.35, -8.35) mm, rotated rx 180 ry 0 rz 0 deg; joints [37.846, -50.454, 135.385, 37.998, -85.131, -2.846]
  MoveC 400 to (267.87, 313.17, -8.35) mm, rotated rx 180 ry 0 rz 0 deg; joints [37.853, -50.465, 135.421, 38.003, -85.151, -2.831] to (268.06, 312.72, -8.35) mm, rotated rx 180 ry 0 rz 0 deg; joints [37.84, -50.474, 135.452, 37.99, -85.168, -2.816]
  MoveL 401 to (268.06, 287.32, -8.35) mm, rotated rx -180 ry 0 rz 0 deg; joints [36.787, -50.788, 136.605, 36.895, -85.782, -2.238]
  MoveL 402 to (217.26, 287.32, -8.35) mm, rotated rx -180 ry 0 rz 0 deg; joints [35.249, -49.835, 133.497, 35.466, -83.96, -3.401]
  MoveL 403 to (217.26, 338.12, -8.35) mm, rotated rx 180 ry 0 rz 0 deg; joints [37.293, -49.146, 131.203, 37.629, -82.822, -4.568]
  MoveL 404 to (268.06, 338.12, -8.35) mm, rotated rx -180 ry 0 rz 0 deg; joints [38.864, -50.138, 134.265, 39.063, -84.562, -3.425]
  MoveL 405 to (268.06, 312.72, -8.35) mm, rotated rx 180 ry 0 rz 0 deg; joints [37.84, -50.474, 135.452, 37.99, -85.168, -2.816]
  MoveC 406 to (267.87, 312.27, -8.35) mm, rotated rx 180 ry 0 rz 0 deg; joints [37.816, -50.476, 135.462, 37.965, -85.172, -2.81] to (267.42, 312.08, -8.35) mm, rotated rx -180 ry 0 rz 0 deg; joints [37.794, -50.471, 135.444, 37.944, -85.161, -2.816]
  MoveL 407 to (266.79, 312.08, -8.35) mm, rotated rx -180 ry 0 rz 0 deg; joints [37.774, -50.459, 135.406, 37.925, -85.139, -2.831]
  MoveC 408 to (266.34, 312.08, -8.16) mm, rotated rx 180 ry 0 rz 0 deg; joints [37.759, -50.466, 135.382, 37.912, -85.114, -2.849] to (266.15, 312.08, -7.72) mm, rotated rx -180 ry 0 rz 0 deg; joints [37.753, -50.498, 135.377, 37.908, -85.085, -2.872]
  Set speed (1000.0 mm/s)
  MoveL 409 to (266.15, 312.08, 6) mm, rotated rx -180 ry 0 rz 0 deg; joints [37.744, -51.588, 135.56, 37.95, -84.368, -3.431]
  MoveL 410 to (139.15, 313.35, 6) mm, rotated rx 180 ry 0 rz 0 deg; joints [34.115, -48.82, 127.555, 34.728, -79.828, -6.118]
  Set speed (25.4 mm/s)
  MoveL 411 to (139.15, 313.35, -3.54) mm, rotated rx -180 ry 0 rz 0 deg; joints [34.121, -48.146, 127.44, 34.678, -80.288, -5.796]
  MoveC 412 to (139.34, 313.35, -3.99) mm, rotated rx 180 ry 0 rz 0 deg; joints [34.126, -48.119, 127.446, 34.68, -80.316, -5.777] to (139.79, 313.35, -4.17) mm, rotated rx 180 ry 0 rz 0 deg; joints [34.138, -48.116, 127.473, 34.689, -80.342, -5.762]
  Set speed (50.8 mm/s)
  MoveL 413 to (140.42, 313.36, -4.18) mm, rotated rx -180 ry 0 rz 0 deg; joints [34.155, -48.131, 127.514, 34.704, -80.366, -5.749]
  MoveC 414 to (140.87, 313.17, -4.17) mm, rotated rx -180 ry 0 rz 0 deg; joints [34.159, -48.144, 127.552, 34.706, -80.386, -5.736] to (141.06, 312.72, -4.17) mm, rotated rx -180 ry 0 rz 0 deg; joints [34.147, -48.155, 127.584, 34.691, -80.402, -5.722]
  MoveL 415 to (141.06, 287.32, -4.17) mm, rotated rx -180 ry 0 rz 0 deg; joints [33.139, -48.518, 128.684, 33.608, -80.912, -5.153]
  MoveL 416 to (90.26, 287.32, -4.17) mm, rotated rx 180 ry 0 rz 0 deg; joints [31.855, -47.305, 125.298, 32.521, -78.958, -6.15]
  MoveL 417 to (90.26, 338.12, -4.17) mm, rotated rx -180 ry 0 rz 0 deg; joints [33.808, -46.534, 123.095, 34.66, -78.003, -7.324]
  MoveL 418 to (141.06, 338.12, -4.18) mm, rotated rx 180 ry 0 rz 0 deg; joints [35.13, -47.772, 126.448, 35.759, -79.894, -6.318]
  MoveL 419 to (141.06, 312.72, -4.17) mm, rotated rx -180 ry 0 rz 0 deg; joints [34.147, -48.155, 127.584, 34.691, -80.402, -5.722]
  MoveC 420 to (140.87, 312.27, -4.18) mm, rotated rx 180 ry 0 rz 0 deg; joints [34.124, -48.157, 127.591, 34.668, -80.404, -5.715] to (140.42, 312.09, -4.18) mm, rotated rx -180 ry 0 rz 0 deg; joints [34.105, -48.149, 127.57, 34.65, -80.391, -5.72]
  MoveL 421 to (139.79, 312.08, -4.17) mm, rotated rx -180 ry 0 rz 0 deg; joints [34.088, -48.134, 127.529, 34.636, -80.367, -5.733]
  MoveC 422 to (139.34, 312.08, -3.99) mm, rotated rx 180 ry 0 rz 0 deg; joints [34.076, -48.137, 127.502, 34.626, -80.342, -5.748] to (139.15, 312.08, -3.54) mm, rotated rx -180 ry 0 rz 0 deg; joints [34.071, -48.165, 127.495, 34.624, -80.313, -5.767]
  Set speed (1000.0 mm/s)
  MoveL 423 to (139.15, 312.08, 5) mm, rotated rx -180 ry 0 rz 0 deg; joints [34.066, -48.768, 127.599, 34.669, -79.901, -6.055]
  MoveL 424 to (139.15, 313.35, 5) mm, rotated rx 180 ry 0 rz 0 deg; joints [34.116, -48.749, 127.543, 34.723, -79.876, -6.084]
  Set speed (25.4 mm/s)
  MoveL 425 to (139.15, 313.36, 1.83) mm, rotated rx -180 ry 0 rz 0 deg; joints [34.117, -48.525, 127.505, 34.706, -80.03, -5.976]
  MoveL 426 to (139.15, 313.36, -7.71) mm, rotated rx -180 ry 0 rz 0 deg; joints [34.123, -47.85, 127.387, 34.657, -80.488, -5.656]
  MoveC 427 to (139.34, 313.36, -8.16) mm, rotated rx -180 ry 0 rz 0 deg; joints [34.128, -47.823, 127.393, 34.659, -80.516, -5.638] to (139.79, 313.36, -8.35) mm, rotated rx 180 ry 0 rz 0 deg; joints [34.14, -47.82, 127.42, 34.669, -80.542, -5.622]
  Set speed (50.8 mm/s)
  MoveL 428 to (140.42, 313.36, -8.35) mm, rotated rx 180 ry 0 rz 0 deg; joints [34.157, -47.835, 127.461, 34.683, -80.565, -5.609]
  MoveC 429 to (140.87, 313.17, -8.35) mm, rotated rx -180 ry 0 rz 0 deg; joints [34.162, -47.848, 127.499, 34.685, -80.586, -5.596] to (141.06, 312.72, -8.35) mm, rotated rx -180 ry 0 rz 0 deg; joints [34.149, -47.858, 127.531, 34.671, -80.602, -5.582]
  MoveL 430 to (141.06, 287.32, -8.35) mm, rotated rx -180 ry 0 rz 0 deg; joints [33.142, -48.217, 128.63, 33.589, -81.117, -5.015]
  MoveL 431 to (90.26, 287.32, -8.35) mm, rotated rx -180 ry 0 rz 0 deg; joints [31.858, -47.018, 125.246, 32.499, -79.156, -6.021]
  MoveL 432 to (90.26, 338.12, -8.35) mm, rotated rx -180 ry 0 rz 0 deg; joints [33.81, -46.255, 123.044, 34.635, -78.191, -7.192]
  MoveL 433 to (141.06, 338.12, -8.35) mm, rotated rx 180 ry 0 rz 0 deg; joints [35.133, -47.481, 126.395, 35.737, -80.089, -6.176]
  MoveL 434 to (141.06, 312.72, -8.35) mm, rotated rx -180 ry 0 rz 0 deg; joints [34.149, -47.858, 127.531, 34.671, -80.602, -5.582]
  MoveC 435 to (140.87, 312.27, -8.35) mm, rotated rx -180 ry 0 rz 0 deg; joints [34.127, -47.861, 127.538, 34.647, -80.604, -5.575] to (140.42, 312.09, -8.35) mm, rotated rx -180 ry 0 rz 0 deg; joints [34.107, -47.853, 127.517, 34.629, -80.591, -5.58]
  MoveL 436 to (139.79, 312.09, -8.35) mm, rotated rx -180 ry 0 rz 0 deg; joints [34.09, -47.839, 127.476, 34.615, -80.567, -5.593]
  MoveC 437 to (139.34, 312.08, -8.16) mm, rotated rx 180 ry 0 rz 0 deg; joints [34.078, -47.841, 127.449, 34.606, -80.542, -5.609] to (139.15, 312.08, -7.72) mm, rotated rx 180 ry 0 rz 0 deg; joints [34.073, -47.869, 127.442, 34.604, -80.513, -5.627]
  Set speed (1000.0 mm/s)
  MoveL 438 to (139.15, 312.08, 6) mm, rotated rx 180 ry 0 rz 0 deg; joints [34.065, -48.839, 127.611, 34.674, -79.853, -6.089]
  MoveL 439 to (139.15, 131.49, 6) mm, rotated rx -180 ry 0 rz 0 deg; joints [26.39, -51.096, 134.631, 26.576, -83.343, -2.615]
  Set speed (25.4 mm/s)
  MoveL 440 to (139.15, 131.49, -3.54) mm, rotated rx -180 ry 0 rz 0 deg; joints [26.396, -50.349, 134.506, 26.55, -83.9, -2.336]
  MoveC 441 to (139.34, 131.48, -3.99) mm, rotated rx -180 ry 0 rz 0 deg; joints [26.4, -50.317, 134.513, 26.553, -83.934, -2.319] to (139.79, 131.49, -4.17) mm, rotated rx 180 ry 0 rz 0 deg; joints [26.41, -50.312, 134.541, 26.562, -83.964, -2.305]
  Set speed (50.8 mm/s)
  MoveL 442 to (140.42, 131.49, -4.18) mm, rotated rx -180 ry 0 rz 0 deg; joints [26.425, -50.326, 134.584, 26.575, -83.991, -2.293]
  MoveC 443 to (140.87, 131.3, -4.17) mm, rotated rx 180 ry 0 rz 0 deg; joints [26.427, -50.337, 134.621, 26.575, -84.014, -2.282] to (141.06, 130.85, -4.17) mm, rotated rx -180 ry 0 rz 0 deg; joints [26.41, -50.345, 134.649, 26.558, -84.031, -2.272]
  MoveL 444 to (141.06, 105.45, -4.18) mm, rotated rx 180 ry 0 rz 0 deg; joints [25.233, -50.578, 135.481, 25.35, -84.522, -1.908]
  MoveL 445 to (90.26, 105.45, -4.17) mm, rotated rx 180 ry 0 rz 0 deg; joints [24.157, -49.467, 131.966, 24.384, -82.291, -2.817]
  MoveL 446 to (90.26, 156.25, -4.18) mm, rotated rx 180 ry 0 rz 0 deg; joints [26.418, -48.954, 130.299, 26.736, -81.387, -3.61]
  MoveL 447 to (141.06, 156.25, -4.18) mm, rotated rx 180 ry 0 rz 0 deg; joints [27.564, -50.095, 133.777, 27.748, -83.533, -2.665]
  MoveL 448 to (141.06, 130.85, -4.17) mm, rotated rx -180 ry 0 rz 0 deg; joints [26.41, -50.345, 134.649, 26.558, -84.031, -2.272]
  MoveC 449 to (140.87, 130.4, -4.18) mm, rotated rx -180 ry 0 rz 0 deg; joints [26.385, -50.345, 134.651, 26.533, -84.032, -2.268] to (140.42, 130.21, -4.18) mm, rotated rx -180 ry 0 rz 0 deg; joints [26.367, -50.338, 134.627, 26.515, -84.016, -2.274]
  MoveL 450 to (139.79, 130.22, -4.17) mm, rotated rx -180 ry 0 rz 0 deg; joints [26.352, -50.324, 134.584, 26.502, -83.989, -2.286]
  MoveC 451 to (139.34, 130.22, -3.99) mm, rotated rx 180 ry 0 rz 0 deg; joints [26.342, -50.329, 134.556, 26.493, -83.959, -2.3] to (139.15, 130.21, -3.54) mm, rotated rx -180 ry 0 rz 0 deg; joints [26.337, -50.361, 134.549, 26.49, -83.925, -2.317]
  Set speed (1000.0 mm/s)
  MoveL 452 to (139.15, 130.22, 5) mm, rotated rx -180 ry 0 rz 0 deg; joints [26.333, -51.03, 134.661, 26.513, -83.426, -2.566]
  MoveL 453 to (139.15, 131.48, 5) mm, rotated rx -180 ry 0 rz 0 deg; joints [26.391, -51.017, 134.618, 26.573, -83.402, -2.586]
  Set speed (25.4 mm/s)
  MoveL 454 to (139.15, 131.49, 1.82) mm, rotated rx -180 ry 0 rz 0 deg; joints [26.393, -50.769, 134.578, 26.564, -83.587, -2.492]
  MoveL 455 to (139.15, 131.48, -7.72) mm, rotated rx -180 ry 0 rz 0 deg; joints [26.398, -50.021, 134.449, 26.54, -84.142, -2.214]
  MoveC 456 to (139.34, 131.48, -8.16) mm, rotated rx 180 ry 0 rz 0 deg; joints [26.403, -49.99, 134.456, 26.543, -84.176, -2.198] to (139.79, 131.48, -8.35) mm, rotated rx 180 ry 0 rz 0 deg; joints [26.413, -49.985, 134.483, 26.552, -84.206, -2.184]
  Set speed (50.8 mm/s)
  MoveL 457 to (140.42, 131.49, -8.35) mm, rotated rx -180 ry 0 rz 0 deg; joints [26.427, -49.998, 134.527, 26.565, -84.233, -2.172]
  MoveC 458 to (140.87, 131.3, -8.35) mm, rotated rx -180 ry 0 rz 0 deg; joints [26.429, -50.009, 134.563, 26.565, -84.256, -2.16] to (141.06, 130.85, -8.35) mm, rotated rx -180 ry 0 rz 0 deg; joints [26.413, -50.017, 134.591, 26.548, -84.273, -2.15]
  MoveL 459 to (141.06, 105.45, -8.35) mm, rotated rx -180 ry 0 rz 0 deg; joints [25.235, -50.245, 135.423, 25.341, -84.769, -1.79]
  MoveL 460 to (90.26, 105.45, -8.35) mm, rotated rx 180 ry 0 rz 0 deg; joints [24.159, -49.152, 131.91, 24.372, -82.527, -2.71]
  MoveL 461 to (90.26, 156.25, -8.35) mm, rotated rx -180 ry 0 rz 0 deg; joints [26.42, -48.646, 130.244, 26.721, -81.613, -3.495]
  MoveL 462 to (141.06, 156.25, -8.35) mm, rotated rx 180 ry 0 rz 0 deg; joints [27.567, -49.771, 133.72, 27.737, -83.769, -2.54]
  MoveL 463 to (141.06, 130.85, -8.35) mm, rotated rx -180 ry 0 rz 0 deg; joints [26.413, -50.017, 134.591, 26.548, -84.273, -2.15]
  MoveC 464 to (140.87, 130.4, -8.35) mm, rotated rx -180 ry 0 rz 0 deg; joints [26.388, -50.017, 134.593, 26.523, -84.274, -2.147] to (140.42, 130.22, -8.35) mm, rotated rx -180 ry 0 rz 0 deg; joints [26.369, -50.01, 134.569, 26.505, -84.258, -2.153]
  MoveL 465 to (139.79, 130.21, -8.35) mm, rotated rx -180 ry 0 rz 0 deg; joints [26.355, -49.996, 134.526, 26.492, -84.231, -2.165]
  MoveC 466 to (139.34, 130.21, -8.16) mm, rotated rx 180 ry 0 rz 0 deg; joints [26.344, -50.002, 134.498, 26.483, -84.201, -2.179] to (139.15, 130.21, -7.72) mm, rotated rx -180 ry 0 rz 0 deg; joints [26.34, -50.033, 134.492, 26.48, -84.167, -2.196]
  Set speed (1000.0 mm/s)
  MoveL 467 to (139.15, 130.21, 6) mm, rotated rx 180 ry 0 rz 0 deg; joints [26.332, -51.108, 134.674, 26.516, -83.367, -2.596]
  MoveL 468 to (266.15, 131.49, 6) mm, rotated rx -180 ry 0 rz 0 deg; joints [29.6, -53.527, 142.984, 29.601, -88.658, 0.004]
  Set speed (25.4 mm/s)
  MoveL 469 to (266.15, 131.48, -3.54) mm, rotated rx 180 ry 0 rz 0 deg; joints [29.606, -52.666, 142.844, 29.601, -89.286, 0.361]
  MoveC 470 to (266.34, 131.49, -3.99) mm, rotated rx -180 ry 0 rz 0 deg; joints [29.611, -52.628, 142.849, 29.606, -89.323, 0.382] to (266.79, 131.48, -4.17) mm, rotated rx 180 ry 0 rz 0 deg; joints [29.624, -52.618, 142.875, 29.618, -89.354, 0.399]
  Set speed (50.8 mm/s)
  MoveL 471 to (267.42, 131.49, -4.18) mm, rotated rx 180 ry 0 rz 0 deg; joints [29.642, -52.627, 142.915, 29.636, -89.38, 0.415]
  MoveC 472 to (267.87, 131.3, -4.17) mm, rotated rx -180 ry 0 rz 0 deg; joints [29.646, -52.635, 142.95, 29.639, -89.404, 0.428] to (268.06, 130.85, -4.17) mm, rotated rx 180 ry 0 rz 0 deg; joints [29.629, -52.641, 142.978, 29.622, -89.423, 0.439]
  MoveL 473 to (268.06, 105.45, -4.17) mm, rotated rx -180 ry 0 rz 0 deg; joints [28.355, -52.815, 143.867, 28.348, -90.056, 0.772]
  MoveL 474 to (217.26, 105.45, -4.17) mm, rotated rx -180 ry 0 rz 0 deg; joints [27.025, -52.02, 140.58, 27.038, -87.848, -0.382]
  MoveL 475 to (217.26, 156.25, -4.18) mm, rotated rx 180 ry 0 rz 0 deg; joints [29.465, -51.598, 138.812, 29.511, -86.706, -1.1]
  MoveL 476 to (268.06, 156.25, -4.17) mm, rotated rx 180 ry 0 rz 0 deg; joints [30.87, -52.448, 142.049, 30.87, -88.788, 0.068]
  MoveL 477 to (268.06, 130.85, -4.17) mm, rotated rx 180 ry 0 rz 0 deg; joints [29.629, -52.641, 142.978, 29.622, -89.423, 0.439]
  MoveC 478 to (267.87, 130.4, -4.18) mm, rotated rx -180 ry 0 rz 0 deg; joints [29.601, -52.642, 142.982, 29.595, -89.426, 0.44] to (267.42, 130.22, -4.18) mm, rotated rx 180 ry 0 rz 0 deg; joints [29.579, -52.636, 142.96, 29.573, -89.412, 0.432]
  MoveL 479 to (266.79, 130.22, -4.17) mm, rotated rx -180 ry 0 rz 0 deg; joints [29.561, -52.627, 142.92, 29.555, -89.385, 0.417]
  MoveC 480 to (266.34, 130.21, -3.99) mm, rotated rx 180 ry 0 rz 0 deg; joints [29.549, -52.637, 142.894, 29.543, -89.354, 0.399] to (266.15, 130.21, -3.54) mm, rotated rx 180 ry 0 rz 0 deg; joints [29.543, -52.675, 142.889, 29.538, -89.317, 0.378]
  Set speed (1000.0 mm/s)
  MoveL 481 to (266.15, 130.22, 5) mm, rotated rx 180 ry 0 rz 0 deg; joints [29.538, -53.447, 143.015, 29.537, -88.755, 0.059]
  MoveL 482 to (266.15, 131.48, 5) mm, rotated rx 180 ry 0 rz 0 deg; joints [29.6, -53.437, 142.97, 29.6, -88.724, 0.041]
  Set speed (25.4 mm/s)
  MoveL 483 to (266.15, 131.49, 1.82) mm, rotated rx 180 ry 0 rz 0 deg; joints [29.602, -53.15, 142.924, 29.6, -88.934, 0.16]
  MoveL 484 to (266.15, 131.48, -7.72) mm, rotated rx 180 ry 0 rz 0 deg; joints [29.609, -52.288, 142.78, 29.602, -89.558, 0.515]
  MoveC 485 to (266.34, 131.49, -8.16) mm, rotated rx 180 ry 0 rz 0 deg; joints [29.614, -52.25, 142.784, 29.607, -89.595, 0.536] to (266.79, 131.48, -8.35) mm, rotated rx -180 ry 0 rz 0 deg; joints [29.627, -52.24, 142.81, 29.62, -89.626, 0.554]
  Set speed (50.8 mm/s)
  MoveL 486 to (267.42, 131.48, -8.35) mm, rotated rx 180 ry 0 rz 0 deg; joints [29.645, -52.249, 142.85, 29.638, -89.653, 0.569]
  MoveC 487 to (267.87, 131.3, -8.35) mm, rotated rx 180 ry 0 rz 0 deg; joints [29.648, -52.257, 142.885, 29.641, -89.676, 0.583] to (268.06, 130.85, -8.35) mm, rotated rx 180 ry 0 rz 0 deg; joints [29.631, -52.263, 142.913, 29.624, -89.696, 0.594]
  MoveL 488 to (268.06, 105.45, -8.35) mm, rotated rx -180 ry 0 rz 0 deg; joints [28.358, -52.431, 143.801, 28.351, -90.337, 0.923]
  MoveL 489 to (217.26, 105.45, -8.35) mm, rotated rx -180 ry 0 rz 0 deg; joints [27.027, -51.658, 140.518, 27.035, -88.115, -0.246]
  MoveL 490 to (217.26, 156.25, -8.35) mm, rotated rx 180 ry 0 rz 0 deg; joints [29.468, -51.247, 138.751, 29.506, -86.958, -0.956]
  MoveL 491 to (268.06, 156.25, -8.35) mm, rotated rx -180 ry 0 rz 0 deg; joints [30.873, -52.076, 141.986, 30.87, -89.053, 0.226]
  MoveL 492 to (268.06, 130.85, -8.35) mm, rotated rx 180 ry 0 rz 0 deg; joints [29.631, -52.263, 142.913, 29.624, -89.696, 0.594]
  MoveC 493 to (267.87, 130.4, -8.35) mm, rotated rx -180 ry 0 rz 0 deg; joints [29.604, -52.263, 142.917, 29.596, -89.699, 0.595] to (267.42, 130.21, -8.35) mm, rotated rx 180 ry 0 rz 0 deg; joints [29.582, -52.258, 142.896, 29.575, -89.685, 0.587]
  MoveL 494 to (266.79, 130.22, -8.35) mm, rotated rx -180 ry 0 rz 0 deg; joints [29.564, -52.249, 142.855, 29.557, -89.658, 0.571]
  MoveC 495 to (266.34, 130.22, -8.16) mm, rotated rx 180 ry 0 rz 0 deg; joints [29.551, -52.259, 142.83, 29.544, -89.627, 0.554] to (266.15, 130.22, -7.72) mm, rotated rx -180 ry 0 rz 0 deg; joints [29.546, -52.297, 142.825, 29.539, -89.59, 0.533]
  Set speed (1000.0 mm/s)
  MoveL 496 to (266.15, 130.21, 6) mm, rotated rx 180 ry 0 rz 0 deg; joints [29.537, -53.538, 143.029, 29.537, -88.688, 0.022]
  MoveL 497 to (393.15, 131.48, 6) mm, rotated rx -180 ry 0 rz 0 deg; joints [33.596, -55.103, 150.756, 33.673, -93.838, 3.403]
  Set speed (25.4 mm/s)
  MoveL 498 to (393.15, 131.49, -3.54) mm, rotated rx -180 ry 0 rz 0 deg; joints [33.604, -54.092, 150.594, 33.715, -94.544, 3.877]
  MoveC 499 to (393.34, 131.49, -3.99) mm, rotated rx 180 ry 0 rz 0 deg; joints [33.611, -54.046, 150.597, 33.724, -94.585, 3.905] to (393.79, 131.49, -4.17) mm, rotated rx -180 ry 0 rz 0 deg; joints [33.627, -54.029, 150.62, 33.742, -94.617, 3.928]
  Set speed (50.8 mm/s)
  MoveL 500 to (394.42, 131.49, -4.18) mm, rotated rx -180 ry 0 rz 0 deg; joints [33.649, -54.034, 150.658, 33.766, -94.643, 3.949]
  MoveC 501 to (394.87, 131.3, -4.18) mm, rotated rx -180 ry 0 rz 0 deg; joints [33.655, -54.037, 150.691, 33.773, -94.667, 3.966] to (395.06, 130.85, -4.17) mm, rotated rx -180 ry 0 rz 0 deg; joints [33.638, -54.04, 150.719, 33.757, -94.69, 3.979]
  MoveL 502 to (395.06, 105.45, -4.17) mm, rotated rx 180 ry 0 rz 0 deg; joints [32.267, -54.102, 151.682, 32.428, -95.537, 4.329]
  MoveL 503 to (344.26, 105.45, -4.18) mm, rotated rx 180 ry 0 rz 0 deg; joints [30.591, -53.72, 148.626, 30.641, -93.353, 2.771]
  MoveL 504 to (344.26, 156.25, -4.18) mm, rotated rx 180 ry 0 rz 0 deg; joints [33.218, -53.466, 146.724, 33.229, -91.856, 2.057]
  MoveL 505 to (395.06, 156.25, -4.17) mm, rotated rx -180 ry 0 rz 0 deg; joints [34.966, -53.953, 149.717, 35.048, -93.854, 3.579]
  MoveL 506 to (395.06, 130.85, -4.17) mm, rotated rx -180 ry 0 rz 0 deg; joints [33.638, -54.04, 150.719, 33.757, -94.69, 3.979]
  MoveC 507 to (394.87, 130.4, -4.17) mm, rotated rx -180 ry 0 rz 0 deg; joints [33.607, -54.04, 150.726, 33.727, -94.697, 3.979] to (394.42, 130.21, -4.17) mm, rotated rx -180 ry 0 rz 0 deg; joints [33.582, -54.038, 150.707, 33.701, -94.685, 3.967]
  MoveL 508 to (393.79, 130.22, -4.18) mm, rotated rx 180 ry 0 rz 0 deg; joints [33.559, -54.033, 150.67, 33.677, -94.659, 3.947]
  MoveC 509 to (393.34, 130.21, -3.99) mm, rotated rx -180 ry 0 rz 0 deg; joints [33.543, -54.05, 150.646, 33.659, -94.627, 3.923] to (393.15, 130.22, -3.54) mm, rotated rx 180 ry 0 rz 0 deg; joints [33.536, -54.096, 150.643, 33.65, -94.586, 3.895]
  Set speed (1000.0 mm/s)
  MoveL 510 to (393.15, 130.21, 5) mm, rotated rx 180 ry 0 rz 0 deg; joints [33.53, -55.002, 150.788, 33.612, -93.953, 3.472]
  MoveL 511 to (393.15, 131.48, 5) mm, rotated rx -180 ry 0 rz 0 deg; joints [33.597, -54.997, 150.739, 33.677, -93.913, 3.453]
  Set speed (25.4 mm/s)
  MoveL 512 to (393.15, 131.49, 1.82) mm, rotated rx 180 ry 0 rz 0 deg; joints [33.6, -54.66, 150.686, 33.691, -94.149, 3.611]
  MoveL 513 to (393.15, 131.48, -7.71) mm, rotated rx 180 ry 0 rz 0 deg; joints [33.607, -53.651, 150.52, 33.735, -94.85, 4.082]
  MoveC 514 to (393.34, 131.49, -8.16) mm, rotated rx 180 ry 0 rz 0 deg; joints [33.614, -53.604, 150.523, 33.745, -94.89, 4.11] to (393.79, 131.49, -8.35) mm, rotated rx -180 ry 0 rz 0 deg; joints [33.63, -53.587, 150.546, 33.763, -94.922, 4.133]
  Set speed (50.8 mm/s)
  MoveL 515 to (394.42, 131.49, -8.35) mm, rotated rx -180 ry 0 rz 0 deg; joints [33.652, -53.591, 150.583, 33.787, -94.948, 4.154]
  MoveC 516 to (394.87, 131.3, -8.35) mm, rotated rx -180 ry 0 rz 0 deg; joints [33.658, -53.595, 150.617, 33.794, -94.973, 4.172] to (395.06, 130.85, -8.35) mm, rotated rx -180 ry 0 rz 0 deg; joints [33.641, -53.597, 150.645, 33.778, -94.996, 4.184]
  MoveL 517 to (395.06, 105.45, -8.35) mm, rotated rx -180 ry 0 rz 0 deg; joints [32.27, -53.649, 151.606, 32.452, -95.854, 4.532]
  MoveL 518 to (344.26, 105.45, -8.35) mm, rotated rx 180 ry 0 rz 0 deg; joints [30.594, -53.297, 148.555, 30.656, -93.656, 2.951]
  MoveL 519 to (344.26, 156.25, -8.35) mm, rotated rx 180 ry 0 rz 0 deg; joints [33.221, -53.059, 146.655, 33.239, -92.139, 2.243]
  MoveL 520 to (395.06, 156.25, -8.35) mm, rotated rx 180 ry 0 rz 0 deg; joints [34.97, -53.519, 149.644, 35.066, -94.148, 3.787]
  MoveL 521 to (395.06, 130.85, -8.35) mm, rotated rx -180 ry 0 rz 0 deg; joints [33.641, -53.597, 150.645, 33.778, -94.996, 4.184]
  MoveC 522 to (394.87, 130.4, -8.35) mm, rotated rx -180 ry 0 rz 0 deg; joints [33.611, -53.597, 150.651, 33.748, -95.003, 4.185] to (394.42, 130.22, -8.35) mm, rotated rx -180 ry 0 rz 0 deg; joints [33.585, -53.595, 150.632, 33.721, -94.991, 4.173]
  MoveL 523 to (393.79, 130.22, -8.35) mm, rotated rx -180 ry 0 rz 0 deg; joints [33.562, -53.591, 150.595, 33.697, -94.965, 4.152]
  MoveC 524 to (393.34, 130.22, -8.16) mm, rotated rx 180 ry 0 rz 0 deg; joints [33.547, -53.608, 150.572, 33.679, -94.933, 4.128] to (393.15, 130.21, -7.72) mm, rotated rx 180 ry 0 rz 0 deg; joints [33.54, -53.654, 150.569, 33.67, -94.892, 4.1]
  Set speed (1000.0 mm/s)
  MoveL 525 to (393.15, 130.22, 6) mm, rotated rx -180 ry 0 rz 0 deg; joints [33.529, -55.108, 150.805, 33.607, -93.878, 3.422]
  MoveL 526 to (393.15, -54.85, 6) mm, rotated rx -180 ry 0 rz 0 deg; joints [22.572, -55.248, 156.847, 22.921, -99.833, 4.764]
  Set speed (25.4 mm/s)
  MoveL 527 to (393.15, -54.85, -3.54) mm, rotated rx 180 ry 0 rz 0 deg; joints [22.579, -54.076, 156.66, 22.998, -100.739, 5.156]
  MoveC 528 to (393.34, -54.85, -3.99) mm, rotated rx -180 ry 0 rz 0 deg; joints [22.585, -54.021, 156.662, 23.007, -100.792, 5.18] to (393.79, -54.85, -4.18) mm, rotated rx 180 ry 0 rz 0 deg; joints [22.597, -53.996, 156.687, 23.023, -100.836, 5.202]
  Set speed (50.8 mm/s)
  MoveL 529 to (394.42, -54.85, -4.18) mm, rotated rx 180 ry 0 rz 0 deg; joints [22.614, -53.994, 156.727, 23.044, -100.873, 5.222]
  MoveC 530 to (394.87, -55.04, -4.17) mm, rotated rx -180 ry 0 rz 0 deg; joints [22.614, -53.992, 156.76, 23.047, -100.906, 5.236] to (395.06, -55.49, -4.17) mm, rotated rx -180 ry 0 rz 0 deg; joints [22.59, -53.99, 156.783, 23.024, -100.931, 5.241]
  MoveL 531 to (395.06, -80.89, -4.18) mm, rotated rx 180 ry 0 rz 0 deg; joints [20.91, -53.912, 157.418, 21.372, -101.736, 5.155]
  MoveL 532 to (344.26, -80.89, -4.18) mm, rotated rx 180 ry 0 rz 0 deg; joints [19.685, -53.999, 154.153, 19.917, -98.688, 3.716]
  MoveL 533 to (344.26, -30.09, -4.17) mm, rotated rx -180 ry 0 rz 0 deg; joints [22.851, -54.008, 152.887, 23.042, -97.309, 3.736]
  MoveL 534 to (395.06, -30.09, -4.18) mm, rotated rx -180 ry 0 rz 0 deg; joints [24.229, -54.056, 156.1, 24.629, -100.103, 5.261]
  MoveL 535 to (395.06, -55.49, -4.17) mm, rotated rx -180 ry 0 rz 0 deg; joints [22.59, -53.99, 156.783, 23.024, -100.931, 5.241]
  MoveC 536 to (394.87, -55.94, -4.17) mm, rotated rx -180 ry 0 rz 0 deg; joints [22.556, -53.99, 156.783, 22.989, -100.935, 5.234] to (394.42, -56.12, -4.18) mm, rotated rx -180 ry 0 rz 0 deg; joints [22.531, -53.991, 156.76, 22.963, -100.914, 5.22]
  MoveL 537 to (393.79, -56.12, -4.18) mm, rotated rx 180 ry 0 rz 0 deg; joints [22.514, -53.993, 156.72, 22.942, -100.877, 5.199]
  MoveC 538 to (393.34, -56.12, -3.99) mm, rotated rx -180 ry 0 rz 0 deg; joints [22.502, -54.017, 156.695, 22.926, -100.833, 5.177] to (393.15, -56.12, -3.54) mm, rotated rx 180 ry 0 rz 0 deg; joints [22.496, -54.073, 156.693, 22.916, -100.779, 5.153]
  Set speed (1000.0 mm/s)
  MoveL 539 to (393.15, -56.12, 5) mm, rotated rx -180 ry 0 rz 0 deg; joints [22.49, -55.122, 156.861, 22.847, -99.968, 4.804]
  MoveL 540 to (393.15, -54.85, 5) mm, rotated rx 180 ry 0 rz 0 deg; joints [22.573, -55.125, 156.828, 22.929, -99.929, 4.805]
  Set speed (25.4 mm/s)
  MoveL 541 to (393.15, -54.85, 1.82) mm, rotated rx -180 ry 0 rz 0 deg; joints [22.575, -54.735, 156.767, 22.954, -100.232, 4.936]
  MoveL 542 to (393.15, -54.85, -7.71) mm, rotated rx -180 ry 0 rz 0 deg; joints [22.582, -53.566, 156.574, 23.033, -101.13, 5.325]
  MoveC 543 to (393.34, -54.85, -8.16) mm, rotated rx 180 ry 0 rz 0 deg; joints [22.588, -53.51, 156.576, 23.043, -101.183, 5.35] to (393.79, -54.85, -8.35) mm, rotated rx -180 ry 0 rz 0 deg; joints [22.6, -53.485, 156.601, 23.059, -101.226, 5.372]
  Set speed (50.8 mm/s)
  MoveL 544 to (394.42, -54.85, -8.35) mm, rotated rx 180 ry 0 rz 0 deg; joints [22.617, -53.483, 156.64, 23.08, -101.264, 5.393]
  MoveC 545 to (394.87, -55.04, -8.35) mm, rotated rx 180 ry 0 rz 0 deg; joints [22.617, -53.48, 156.674, 23.083, -101.297, 5.407] to (395.06, -55.49, -8.35) mm, rotated rx 180 ry 0 rz 0 deg; joints [22.593, -53.478, 156.697, 23.06, -101.323, 5.412]
  MoveL 546 to (395.06, -80.89, -8.35) mm, rotated rx -180 ry 0 rz 0 deg; joints [20.913, -53.391, 157.33, 21.408, -102.139, 5.317]
  MoveL 547 to (344.26, -80.89, -8.35) mm, rotated rx 180 ry 0 rz 0 deg; joints [19.688, -53.519, 154.072, 19.941, -99.062, 3.854]
  MoveL 548 to (344.26, -30.09, -8.35) mm, rotated rx -180 ry 0 rz 0 deg; joints [22.854, -53.542, 152.808, 23.064, -97.665, 3.889]
  MoveL 549 to (395.06, -30.09, -8.35) mm, rotated rx -180 ry 0 rz 0 deg; joints [24.233, -53.553, 156.015, 24.664, -100.483, 5.439]
  MoveL 550 to (395.06, -55.49, -8.35) mm, rotated rx 180 ry 0 rz 0 deg; joints [22.593, -53.478, 156.697, 23.06, -101.323, 5.412]
  MoveC 551 to (394.87, -55.94, -8.35) mm, rotated rx 180 ry 0 rz 0 deg; joints [22.559, -53.477, 156.697, 23.025, -101.326, 5.405] to (394.42, -56.12, -8.35) mm, rotated rx 180 ry 0 rz 0 deg; joints [22.534, -53.479, 156.673, 22.998, -101.305, 5.39]
  MoveL 552 to (393.79, -56.12, -8.35) mm, rotated rx -180 ry 0 rz 0 deg; joints [22.517, -53.481, 156.633, 22.978, -101.268, 5.369]
  MoveC 553 to (393.34, -56.12, -8.16) mm, rotated rx 180 ry 0 rz 0 deg; joints [22.505, -53.506, 156.609, 22.961, -101.224, 5.347] to (393.15, -56.12, -7.72) mm, rotated rx 180 ry 0 rz 0 deg; joints [22.499, -53.562, 156.607, 22.951, -101.171, 5.323]
  Set speed (1000.0 mm/s)
  MoveL 554 to (393.15, -56.12, 6) mm, rotated rx -180 ry 0 rz 0 deg; joints [22.489, -55.246, 156.88, 22.839, -99.872, 4.763]
  MoveL 555 to (266.15, -54.85, 6) mm, rotated rx 180 ry 0 rz 0 deg; joints [19.569, -54.526, 148.561, 19.589, -92.933, 1.624]
  Set speed (25.4 mm/s)
  MoveL 556 to (266.15, -54.85, -3.54) mm, rotated rx -180 ry 0 rz 0 deg; joints [19.575, -53.562, 148.406, 19.611, -93.694, 1.896]
  MoveC 557 to (266.34, -54.85, -3.99) mm, rotated rx -180 ry 0 rz 0 deg; joints [19.579, -53.518, 148.41, 19.616, -93.739, 1.913] to (266.79, -54.85, -4.18) mm, rotated rx 180 ry 0 rz 0 deg; joints [19.588, -53.504, 148.437, 19.626, -93.778, 1.928]
  Set speed (50.8 mm/s)
  MoveL 558 to (267.42, -54.85, -4.18) mm, rotated rx -180 ry 0 rz 0 deg; joints [19.601, -53.511, 148.48, 19.64, -93.812, 1.941]
  MoveC 559 to (267.87, -55.04, -4.17) mm, rotated rx 180 ry 0 rz 0 deg; joints [19.6, -53.515, 148.514, 19.639, -93.839, 1.951] to (268.06, -55.49, -4.18) mm, rotated rx 180 ry 0 rz 0 deg; joints [19.578, -53.518, 148.537, 19.617, -93.859, 1.956]
  MoveL 560 to (268.06, -80.89, -4.17) mm, rotated rx -180 ry 0 rz 0 deg; joints [18.087, -53.576, 149.113, 18.136, -94.394, 1.994]
  MoveL 561 to (217.26, -80.89, -4.17) mm, rotated rx 180 ry 0 rz 0 deg; joints [17.154, -53.002, 145.662, 17.155, -91.673, 1.057]
  MoveL 562 to (217.26, -30.09, -4.18) mm, rotated rx -180 ry 0 rz 0 deg; joints [19.98, -52.814, 144.505, 19.975, -90.72, 0.85]
  MoveL 563 to (268.06, -30.09, -4.17) mm, rotated rx 180 ry 0 rz 0 deg; joints [21.041, -53.448, 147.916, 21.071, -93.3, 1.877]
  MoveL 564 to (268.06, -55.49, -4.18) mm, rotated rx 180 ry 0 rz 0 deg; joints [19.578, -53.518, 148.537, 19.617, -93.859, 1.956]
  MoveC 565 to (267.87, -55.94, -4.17) mm, rotated rx -180 ry 0 rz 0 deg; joints [19.548, -53.518, 148.535, 19.587, -93.859, 1.953] to (267.42, -56.12, -4.17) mm, rotated rx -180 ry 0 rz 0 deg; joints [19.528, -53.514, 148.51, 19.567, -93.839, 1.944]
  MoveL 566 to (266.79, -56.12, -4.17) mm, rotated rx -180 ry 0 rz 0 deg; joints [19.515, -53.507, 148.467, 19.553, -93.805, 1.931]
  MoveC 567 to (266.34, -56.12, -3.99) mm, rotated rx -180 ry 0 rz 0 deg; joints [19.505, -53.522, 148.44, 19.543, -93.767, 1.916] to (266.15, -56.12, -3.54) mm, rotated rx 180 ry 0 rz 0 deg; joints [19.501, -53.565, 148.435, 19.537, -93.721, 1.9]
  Set speed (1000.0 mm/s)
  MoveL 568 to (266.15, -56.12, 5) mm, rotated rx -180 ry 0 rz 0 deg; joints [19.496, -54.428, 148.575, 19.518, -93.039, 1.657]
  MoveL 569 to (266.15, -54.85, 5) mm, rotated rx 180 ry 0 rz 0 deg; joints [19.57, -54.425, 148.545, 19.592, -93.013, 1.653]
  Set speed (25.4 mm/s)
  MoveL 570 to (266.15, -54.85, 1.82) mm, rotated rx -180 ry 0 rz 0 deg; joints [19.572, -54.104, 148.494, 19.598, -93.267, 1.744]
  MoveL 571 to (266.15, -54.85, -7.71) mm, rotated rx 180 ry 0 rz 0 deg; joints [19.577, -53.141, 148.334, 19.621, -94.024, 2.014]
  MoveC 572 to (266.34, -54.85, -8.16) mm, rotated rx -180 ry 0 rz 0 deg; joints [19.581, -53.097, 148.339, 19.626, -94.069, 2.031] to (266.79, -54.85, -8.35) mm, rotated rx 180 ry 0 rz 0 deg; joints [19.591, -53.083, 148.366, 19.637, -94.107, 2.046]
  Set speed (50.8 mm/s)
  MoveL 573 to (267.42, -54.85, -8.35) mm, rotated rx -180 ry 0 rz 0 deg; joints [19.604, -53.089, 148.408, 19.651, -94.141, 2.059]
